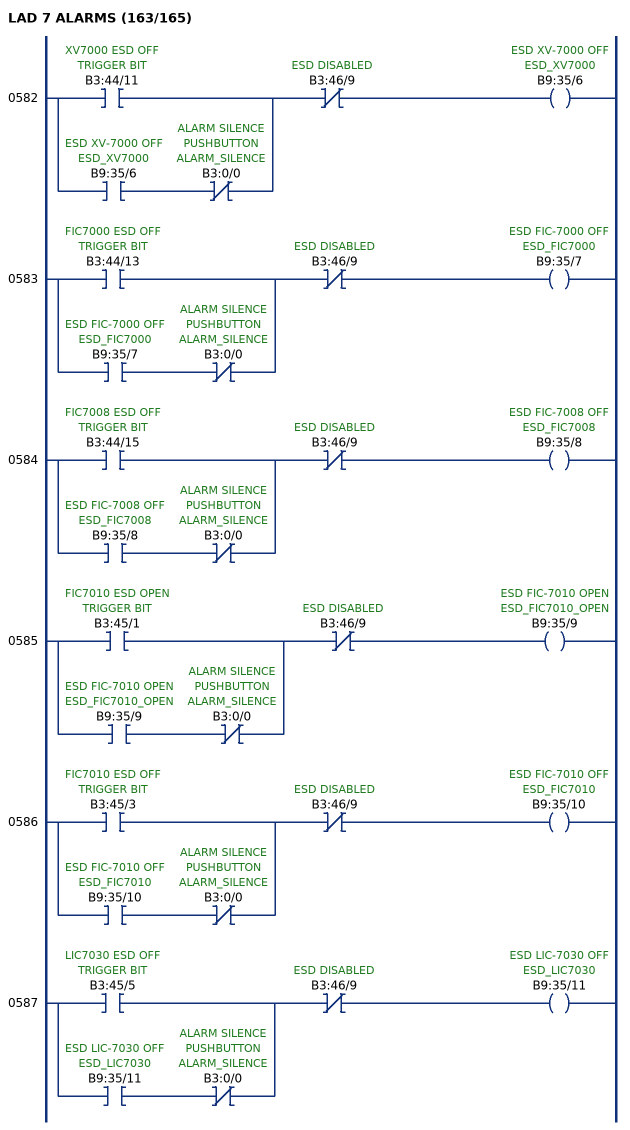
% Rung: 582 %
SOR BST XIC B3:44/11 NXB XIC B9:35/6 XIO B3:0/0 BND XIO B3:46/9 OTE B9:35/6 EOR
%   B3:44/11  "XV7000 ESD OFF TRIGGER BIT" %
%   B9:35/6  ESD_XV7000  "ESD XV-7000 OFF" %
%   B3:0/0  ALARM_SILENCE  "ALARM SILENCE PUSHBUTTON" %
%   B3:46/9  "ESD DISABLED" %
% Rung: 583 %
SOR BST XIC B3:44/13 NXB XIC B9:35/7 XIO B3:0/0 BND XIO B3:46/9 OTE B9:35/7 EOR
%   B3:44/13  "FIC7000 ESD OFF TRIGGER BIT" %
%   B9:35/7  ESD_FIC7000  "ESD FIC-7000 OFF" %
%   B3:0/0  ALARM_SILENCE  "ALARM SILENCE PUSHBUTTON" %
%   B3:46/9  "ESD DISABLED" %
% Rung: 584 %
SOR BST XIC B3:44/15 NXB XIC B9:35/8 XIO B3:0/0 BND XIO B3:46/9 OTE B9:35/8 EOR
%   B3:44/15  "FIC7008 ESD OFF TRIGGER BIT" %
%   B9:35/8  ESD_FIC7008  "ESD FIC-7008 OFF" %
%   B3:0/0  ALARM_SILENCE  "ALARM SILENCE PUSHBUTTON" %
%   B3:46/9  "ESD DISABLED" %
% Rung: 585 %
SOR BST XIC B3:45/1 NXB XIC B9:35/9 XIO B3:0/0 BND XIO B3:46/9 OTE B9:35/9 EOR
%   B3:45/1  "FIC7010 ESD OPEN TRIGGER BIT" %
%   B9:35/9  ESD_FIC7010_OPEN  "ESD FIC-7010 OPEN" %
%   B3:0/0  ALARM_SILENCE  "ALARM SILENCE PUSHBUTTON" %
%   B3:46/9  "ESD DISABLED" %
% Rung: 586 %
SOR BST XIC B3:45/3 NXB XIC B9:35/10 XIO B3:0/0 BND XIO B3:46/9 OTE B9:35/10 EOR
%   B3:45/3  "FIC7010 ESD OFF TRIGGER BIT" %
%   B9:35/10  ESD_FIC7010  "ESD FIC-7010 OFF" %
%   B3:0/0  ALARM_SILENCE  "ALARM SILENCE PUSHBUTTON" %
%   B3:46/9  "ESD DISABLED" %
% Rung: 587 %
SOR BST XIC B3:45/5 NXB XIC B9:35/11 XIO B3:0/0 BND XIO B3:46/9 OTE B9:35/11 EOR
%   B3:45/5  "LIC7030 ESD OFF TRIGGER BIT" %
%   B9:35/11  ESD_LIC7030  "ESD LIC-7030 OFF" %
%   B3:0/0  ALARM_SILENCE  "ALARM SILENCE PUSHBUTTON" %
%   B3:46/9  "ESD DISABLED" %

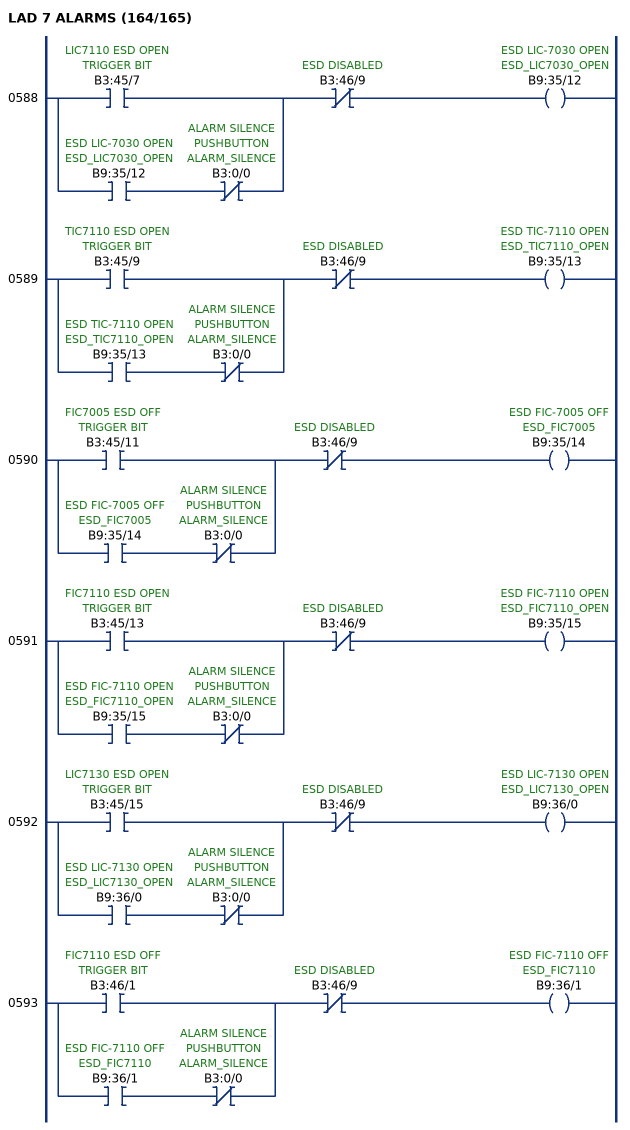
% Rung: 588 %
SOR BST XIC B3:45/7 NXB XIC B9:35/12 XIO B3:0/0 BND XIO B3:46/9 OTE B9:35/12 EOR
%   B3:45/7  "LIC7110 ESD OPEN TRIGGER BIT" %
%   B9:35/12  ESD_LIC7030_OPEN  "ESD LIC-7030 OPEN" %
%   B3:0/0  ALARM_SILENCE  "ALARM SILENCE PUSHBUTTON" %
%   B3:46/9  "ESD DISABLED" %
% Rung: 589 %
SOR BST XIC B3:45/9 NXB XIC B9:35/13 XIO B3:0/0 BND XIO B3:46/9 OTE B9:35/13 EOR
%   B3:45/9  "TIC7110 ESD OPEN TRIGGER BIT" %
%   B9:35/13  ESD_TIC7110_OPEN  "ESD TIC-7110 OPEN" %
%   B3:0/0  ALARM_SILENCE  "ALARM SILENCE PUSHBUTTON" %
%   B3:46/9  "ESD DISABLED" %
% Rung: 590 %
SOR BST XIC B3:45/11 NXB XIC B9:35/14 XIO B3:0/0 BND XIO B3:46/9 OTE B9:35/14 EOR
%   B3:45/11  "FIC7005 ESD OFF TRIGGER BIT" %
%   B9:35/14  ESD_FIC7005  "ESD FIC-7005 OFF" %
%   B3:0/0  ALARM_SILENCE  "ALARM SILENCE PUSHBUTTON" %
%   B3:46/9  "ESD DISABLED" %
% Rung: 591 %
SOR BST XIC B3:45/13 NXB XIC B9:35/15 XIO B3:0/0 BND XIO B3:46/9 OTE B9:35/15 EOR
%   B3:45/13  "FIC7110 ESD OPEN TRIGGER BIT" %
%   B9:35/15  ESD_FIC7110_OPEN  "ESD FIC-7110 OPEN" %
%   B3:0/0  ALARM_SILENCE  "ALARM SILENCE PUSHBUTTON" %
%   B3:46/9  "ESD DISABLED" %
% Rung: 592 %
SOR BST XIC B3:45/15 NXB XIC B9:36/0 XIO B3:0/0 BND XIO B3:46/9 OTE B9:36/0 EOR
%   B3:45/15  "LIC7130 ESD OPEN TRIGGER BIT" %
%   B9:36/0  ESD_LIC7130_OPEN  "ESD LIC-7130 OPEN" %
%   B3:0/0  ALARM_SILENCE  "ALARM SILENCE PUSHBUTTON" %
%   B3:46/9  "ESD DISABLED" %
% Rung: 593 %
SOR BST XIC B3:46/1 NXB XIC B9:36/1 XIO B3:0/0 BND XIO B3:46/9 OTE B9:36/1 EOR
%   B3:46/1  "FIC7110 ESD OFF TRIGGER BIT" %
%   B9:36/1  ESD_FIC7110  "ESD FIC-7110 OFF" %
%   B3:0/0  ALARM_SILENCE  "ALARM SILENCE PUSHBUTTON" %
%   B3:46/9  "ESD DISABLED" %

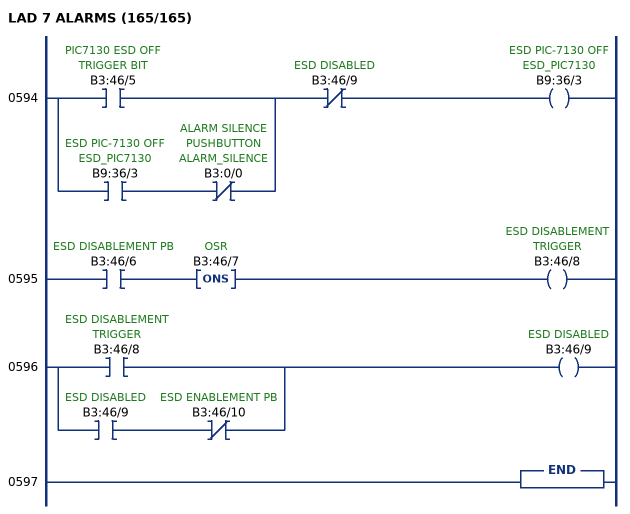
% Rung: 594 %
SOR BST XIC B3:46/5 NXB XIC B9:36/3 XIO B3:0/0 BND XIO B3:46/9 OTE B9:36/3 EOR
%   B3:46/5  "PIC7130 ESD OFF TRIGGER BIT" %
%   B9:36/3  ESD_PIC7130  "ESD PIC-7130 OFF" %
%   B3:0/0  ALARM_SILENCE  "ALARM SILENCE PUSHBUTTON" %
%   B3:46/9  "ESD DISABLED" %
% Rung: 595 %
SOR XIC B3:46/6 OSR B3:46/7 OTE B3:46/8 EOR
%   B3:46/6  "ESD DISABLEMENT PB" %
%   B3:46/7  "OSR" %
%   B3:46/8  "ESD DISABLEMENT TRIGGER" %
% Rung: 596 %
SOR BST XIC B3:46/8 NXB XIC B3:46/9 XIO B3:46/10 BND OTE B3:46/9 EOR
%   B3:46/8  "ESD DISABLEMENT TRIGGER" %
%   B3:46/9  "ESD DISABLED" %
%   B3:46/10  "ESD ENABLEMENT PB" %
% Rung: 597 %
SOR END EOR

LADDER 8 "HMI IO"
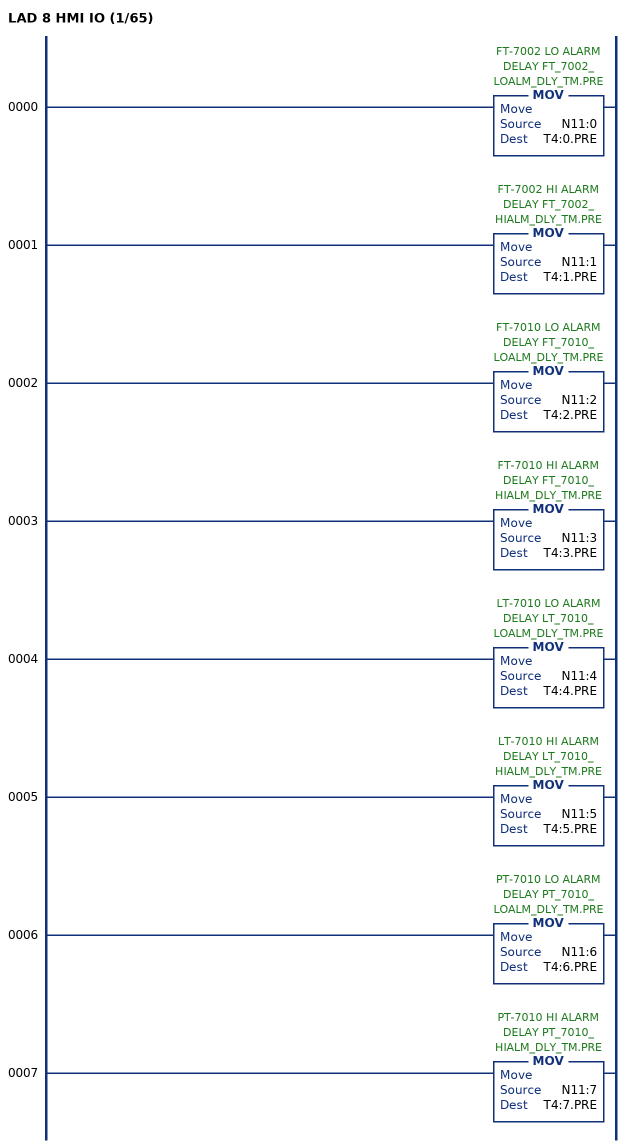
% Rung: 0 %
SOR MOV N11:0 T4:0.PRE EOR
%   N11:0  FT_7002_LOALM_DLY_SP  "FT-7002 LO ALARM DELAY SP FROM HMI" %
%   T4:0  FT_7002_LOALM_DLY_TM  "FT-7002 LO ALARM DELAY" %
% Rung: 1 %
SOR MOV N11:1 T4:1.PRE EOR
%   N11:1  FT_7002_HIALM_DLY_SP  "FT-7002 HI ALARM DELAY SP FROM HMI" %
%   T4:1  FT_7002_HIALM_DLY_TM  "FT-7002 HI ALARM DELAY" %
% Rung: 2 %
SOR MOV N11:2 T4:2.PRE EOR
%   N11:2  FT_7010_LOALM_DLY_SP  "FT-7010 LO ALARM DELAY SP FROM HMI" %
%   T4:2  FT_7010_LOALM_DLY_TM  "FT-7010 LO ALARM DELAY" %
% Rung: 3 %
SOR MOV N11:3 T4:3.PRE EOR
%   N11:3  FT_7010_HIALM_DLY_SP  "FT-7010 HI ALARM DELAY SP FROM HMI" %
%   T4:3  FT_7010_HIALM_DLY_TM  "FT-7010 HI ALARM DELAY" %
% Rung: 4 %
SOR MOV N11:4 T4:4.PRE EOR
%   N11:4  LT_7010_LOALM_DLY_SP  "LT-7010 LO ALARM DELAY SP FROM HMI" %
%   T4:4  LT_7010_LOALM_DLY_TM  "LT-7010 LO ALARM DELAY" %
% Rung: 5 %
SOR MOV N11:5 T4:5.PRE EOR
%   N11:5  LT_7010_HIALM_DLY_SP  "LT-7010 HI ALARM DELAY SP FROM HMI" %
%   T4:5  LT_7010_HIALM_DLY_TM  "LT-7010 HI ALARM DELAY" %
% Rung: 6 %
SOR MOV N11:6 T4:6.PRE EOR
%   N11:6  PT_7010_LOALM_DLY_SP  "PT-7010 LO ALARM DELAY SP FROM HMI" %
%   T4:6  PT_7010_LOALM_DLY_TM  "PT-7010 LO ALARM DELAY" %
% Rung: 7 %
SOR MOV N11:7 T4:7.PRE EOR
%   N11:7  PT_7010_HIALM_DLY_SP  "PT-7010 HI ALARM DELAY SP FROM HMI" %
%   T4:7  PT_7010_HIALM_DLY_TM  "PT-7010 HI ALARM DELAY" %

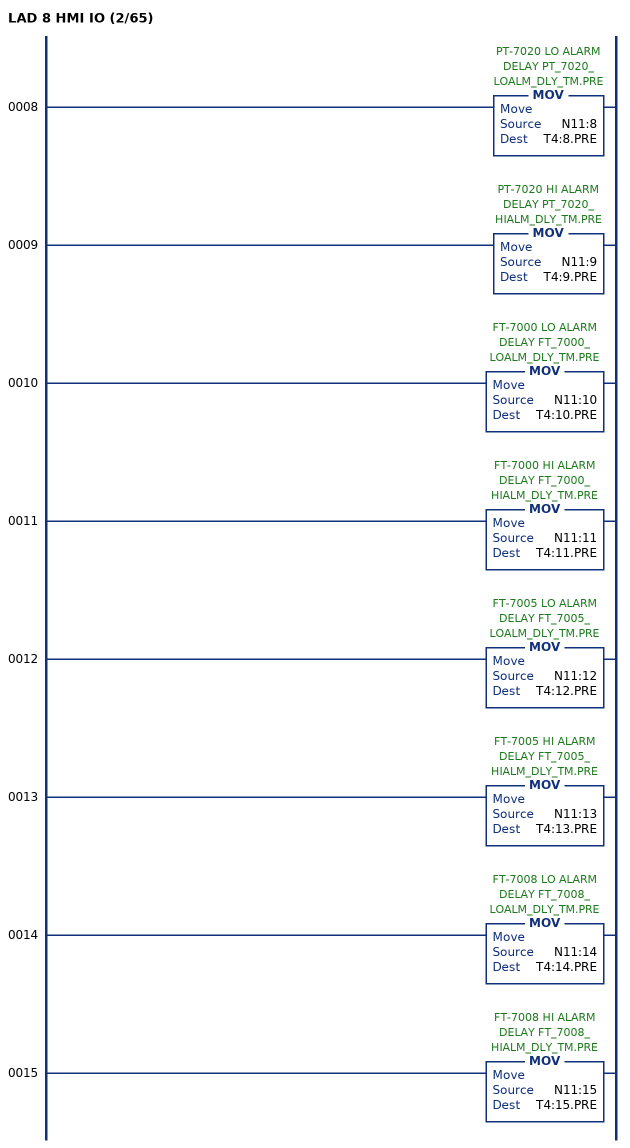
% Rung: 8 %
SOR MOV N11:8 T4:8.PRE EOR
%   N11:8  PT_7020_LOALM_DLY_SP  "PT-7020 LO ALARM DELAY SP FROM HMI" %
%   T4:8  PT_7020_LOALM_DLY_TM  "PT-7020 LO ALARM DELAY" %
% Rung: 9 %
SOR MOV N11:9 T4:9.PRE EOR
%   N11:9  PT_7020_HIALM_DLY_SP  "PT-7020 HI ALARM DELAY SP FROM HMI" %
%   T4:9  PT_7020_HIALM_DLY_TM  "PT-7020 HI ALARM DELAY" %
% Rung: 10 %
SOR MOV N11:10 T4:10.PRE EOR
%   N11:10  FT_7000_LOALM_DLY_SP  "FT-7000 LO ALARM DELAY SP FROM HMI" %
%   T4:10  FT_7000_LOALM_DLY_TM  "FT-7000 LO ALARM DELAY" %
% Rung: 11 %
SOR MOV N11:11 T4:11.PRE EOR
%   N11:11  FT_7000_HIALM_DLY_SP  "FT-7000 HI ALARM DELAY SP FROM HMI" %
%   T4:11  FT_7000_HIALM_DLY_TM  "FT-7000 HI ALARM DELAY" %
% Rung: 12 %
SOR MOV N11:12 T4:12.PRE EOR
%   N11:12  FT_7005_LOALM_DLY_SP  "FT-7005 LO ALARM DELAY SP FROM HMI" %
%   T4:12  FT_7005_LOALM_DLY_TM  "FT-7005 LO ALARM DELAY" %
% Rung: 13 %
SOR MOV N11:13 T4:13.PRE EOR
%   N11:13  FT_7005_HIALM_DLY_SP  "FT-7005 HI ALARM DELAY SP FROM HMI" %
%   T4:13  FT_7005_HIALM_DLY_TM  "FT-7005 HI ALARM DELAY" %
% Rung: 14 %
SOR MOV N11:14 T4:14.PRE EOR
%   N11:14  FT_7008_LOALM_DLY_SP  "FT-7008 LO ALARM DELAY SP FROM HMI" %
%   T4:14  FT_7008_LOALM_DLY_TM  "FT-7008 LO ALARM DELAY" %
% Rung: 15 %
SOR MOV N11:15 T4:15.PRE EOR
%   N11:15  FT_7008_HIALM_DLY_SP  "FT-7008 HI ALARM DELAY SP FROM HMI" %
%   T4:15  FT_7008_HIALM_DLY_TM  "FT-7008 HI ALARM DELAY" %

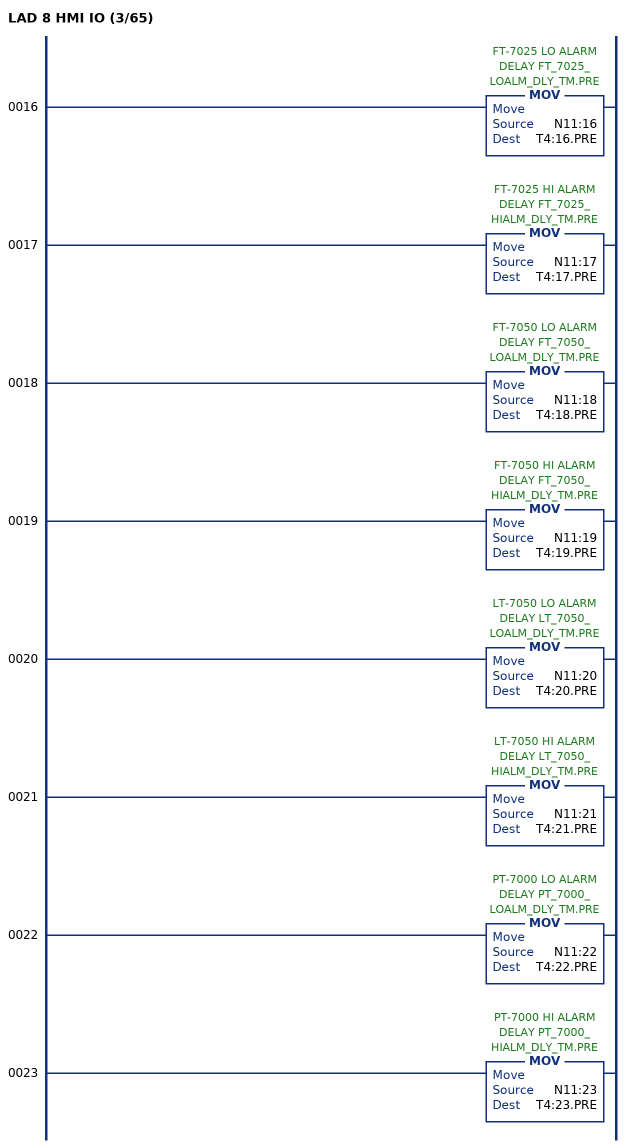
% Rung: 16 %
SOR MOV N11:16 T4:16.PRE EOR
%   N11:16  FT_7025_LOALM_DLY_SP  "FT-7025 LO ALARM DELAY SP FROM HMI" %
%   T4:16  FT_7025_LOALM_DLY_TM  "FT-7025 LO ALARM DELAY" %
% Rung: 17 %
SOR MOV N11:17 T4:17.PRE EOR
%   N11:17  FT_7025_HIALM_DLY_SP  "FT-7025 HI ALARM DELAY SP FROM HMI" %
%   T4:17  FT_7025_HIALM_DLY_TM  "FT-7025 HI ALARM DELAY" %
% Rung: 18 %
SOR MOV N11:18 T4:18.PRE EOR
%   N11:18  FT_7050_LOALM_DLY_SP  "FT-7050 LO ALARM DELAY SP FROM HMI" %
%   T4:18  FT_7050_LOALM_DLY_TM  "FT-7050 LO ALARM DELAY" %
% Rung: 19 %
SOR MOV N11:19 T4:19.PRE EOR
%   N11:19  FT_7050_HIALM_DLY_SP  "FT-7050 HI ALARM DELAY SP FROM HMI" %
%   T4:19  FT_7050_HIALM_DLY_TM  "FT-7050 HI ALARM DELAY" %
% Rung: 20 %
SOR MOV N11:20 T4:20.PRE EOR
%   N11:20  LT_7050_LOALM_DLY_SP  "LT-7050 LO ALARM DELAY SP FROM HMI" %
%   T4:20  LT_7050_LOALM_DLY_TM  "LT-7050 LO ALARM DELAY" %
% Rung: 21 %
SOR MOV N11:21 T4:21.PRE EOR
%   N11:21  LT_7050_HIALM_DLY_SP  "LT-7050 HI ALARM DELAY SP FROM HMI" %
%   T4:21  LT_7050_HIALM_DLY_TM  "LT-7050 HI ALARM DELAY" %
% Rung: 22 %
SOR MOV N11:22 T4:22.PRE EOR
%   N11:22  PT_7000_LOALM_DLY_SP  "PT-7000 LO ALARM DELAY SP FROM HMI" %
%   T4:22  PT_7000_LOALM_DLY_TM  "PT-7000 LO ALARM DELAY" %
% Rung: 23 %
SOR MOV N11:23 T4:23.PRE EOR
%   N11:23  PT_7000_HIALM_DLY_SP  "PT-7000 HI ALARM DELAY SP FROM HMI" %
%   T4:23  PT_7000_HIALM_DLY_TM  "PT-7000 HI ALARM DELAY" %

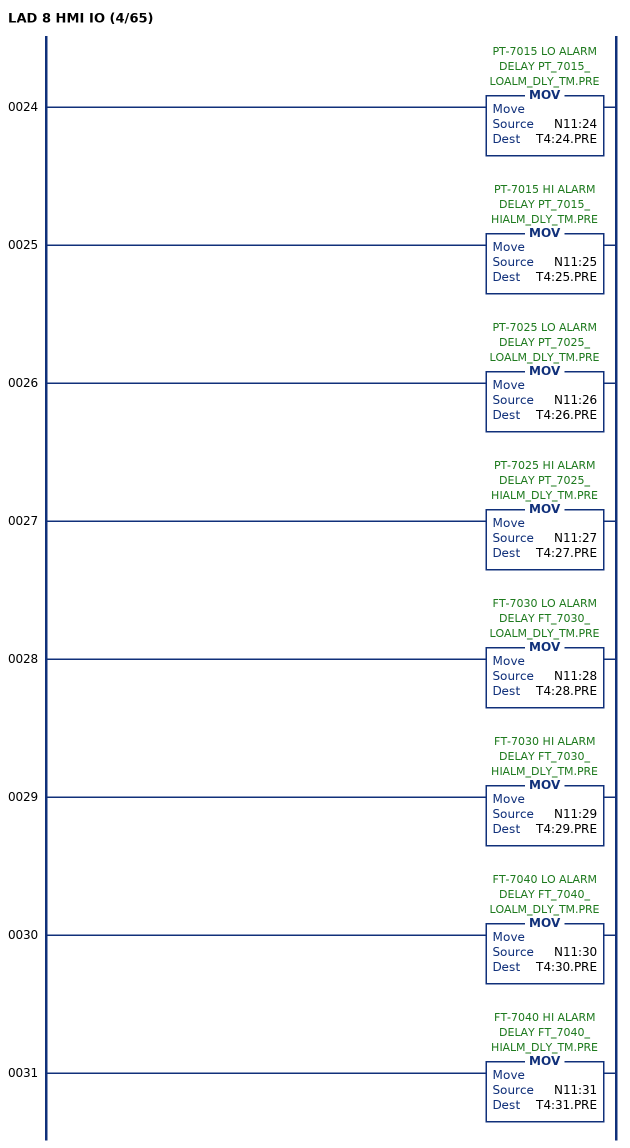
% Rung: 24 %
SOR MOV N11:24 T4:24.PRE EOR
%   N11:24  PT_7015_LOALM_DLY_SP  "PT-7015 LO ALARM DELAY SP FROM HMI" %
%   T4:24  PT_7015_LOALM_DLY_TM  "PT-7015 LO ALARM DELAY" %
% Rung: 25 %
SOR MOV N11:25 T4:25.PRE EOR
%   N11:25  PT_7015_HIALM_DLY_SP  "PT-7015 HI ALARM DELAY SP FROM HMI" %
%   T4:25  PT_7015_HIALM_DLY_TM  "PT-7015 HI ALARM DELAY" %
% Rung: 26 %
SOR MOV N11:26 T4:26.PRE EOR
%   N11:26  PT_7025_LOALM_DLY_SP  "PT-7025 LO ALARM DELAY SP FROM HMI" %
%   T4:26  PT_7025_LOALM_DLY_TM  "PT-7025 LO ALARM DELAY" %
% Rung: 27 %
SOR MOV N11:27 T4:27.PRE EOR
%   N11:27  PT_7025_HIALM_DLY_SP  "PT-7025 HI ALARM DELAY SP FROM HMI" %
%   T4:27  PT_7025_HIALM_DLY_TM  "PT-7025 HI ALARM DELAY" %
% Rung: 28 %
SOR MOV N11:28 T4:28.PRE EOR
%   N11:28  FT_7030_LOALM_DLY_SP  "FT-7030 LO ALARM DELAY SP FROM HMI" %
%   T4:28  FT_7030_LOALM_DLY_TM  "FT-7030 LO ALARM DELAY" %
% Rung: 29 %
SOR MOV N11:29 T4:29.PRE EOR
%   N11:29  FT_7030_HIALM_DLY_SP  "FT-7030 HI ALARM DELAY SP FROM HMI" %
%   T4:29  FT_7030_HIALM_DLY_TM  "FT-7030 HI ALARM DELAY" %
% Rung: 30 %
SOR MOV N11:30 T4:30.PRE EOR
%   N11:30  FT_7040_LOALM_DLY_SP  "FT-7040 LO ALARM DELAY SP FROM HMI" %
%   T4:30  FT_7040_LOALM_DLY_TM  "FT-7040 LO ALARM DELAY" %
% Rung: 31 %
SOR MOV N11:31 T4:31.PRE EOR
%   N11:31  FT_7040_HIALM_DLY_SP  "FT-7040 HI ALARM DELAY SP FROM HMI" %
%   T4:31  FT_7040_HIALM_DLY_TM  "FT-7040 HI ALARM DELAY" %

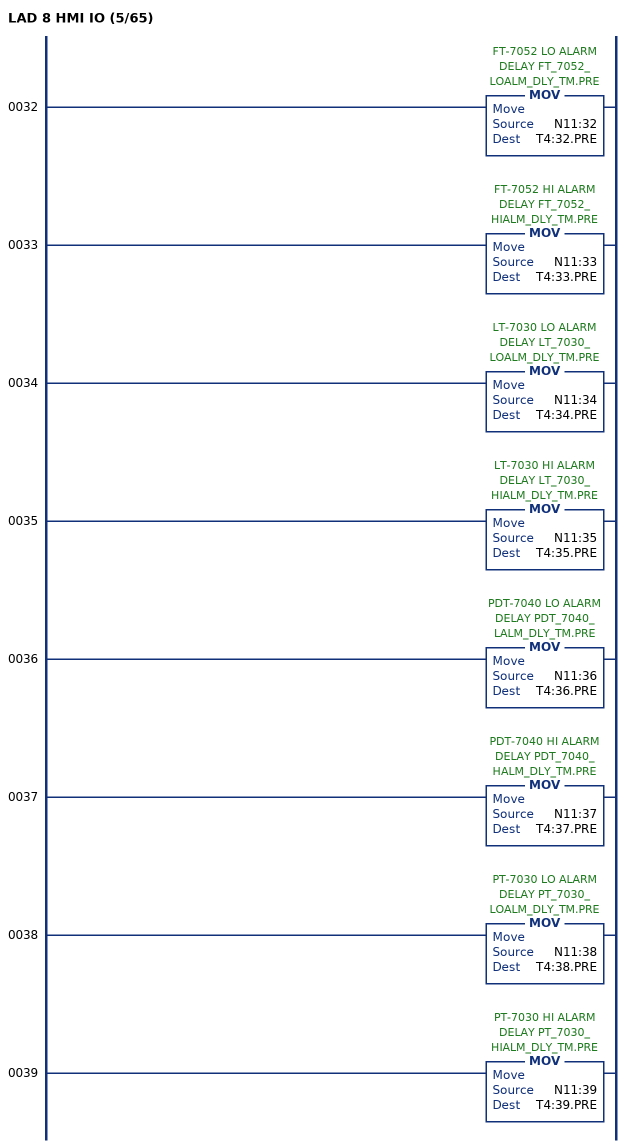
% Rung: 32 %
SOR MOV N11:32 T4:32.PRE EOR
%   N11:32  FT_7052_LOALM_DLY_SP  "FT-7052 LO ALARM DELAY SP FROM HMI" %
%   T4:32  FT_7052_LOALM_DLY_TM  "FT-7052 LO ALARM DELAY" %
% Rung: 33 %
SOR MOV N11:33 T4:33.PRE EOR
%   N11:33  FT_7052_HIALM_DLY_SP  "FT-7052 HI ALARM DELAY SP FROM HMI" %
%   T4:33  FT_7052_HIALM_DLY_TM  "FT-7052 HI ALARM DELAY" %
% Rung: 34 %
SOR MOV N11:34 T4:34.PRE EOR
%   N11:34  LT_7030_LOALM_DLY_SP  "LT-7030 LO ALARM DELAY SP FROM HMI" %
%   T4:34  LT_7030_LOALM_DLY_TM  "LT-7030 LO ALARM DELAY" %
% Rung: 35 %
SOR MOV N11:35 T4:35.PRE EOR
%   N11:35  LT_7030_HIALM_DLY_SP  "LT-7030 HI ALARM DELAY SP FROM HMI" %
%   T4:35  LT_7030_HIALM_DLY_TM  "LT-7030 HI ALARM DELAY" %
% Rung: 36 %
SOR MOV N11:36 T4:36.PRE EOR
%   N11:36  PDT_7040_LALM_DLY_SP  "PDT-7040 LO ALARM DELAY SP FROM HMI" %
%   T4:36  PDT_7040_LALM_DLY_TM  "PDT-7040 LO ALARM DELAY" %
% Rung: 37 %
SOR MOV N11:37 T4:37.PRE EOR
%   N11:37  PDT_7040_HALM_DLY_SP  "PDT-7040 HI ALARM DELAY SP FROM HMI" %
%   T4:37  PDT_7040_HALM_DLY_TM  "PDT-7040 HI ALARM DELAY" %
% Rung: 38 %
SOR MOV N11:38 T4:38.PRE EOR
%   N11:38  PT_7030_LOALM_DLY_SP  "PT-7030 LO ALARM DELAY SP FROM HMI" %
%   T4:38  PT_7030_LOALM_DLY_TM  "PT-7030 LO ALARM DELAY" %
% Rung: 39 %
SOR MOV N11:39 T4:39.PRE EOR
%   N11:39  PT_7030_HIALM_DLY_SP  "PT-7030 HI ALARM DELAY SP FROM HMI" %
%   T4:39  PT_7030_HIALM_DLY_TM  "PT-7030 HI ALARM DELAY" %

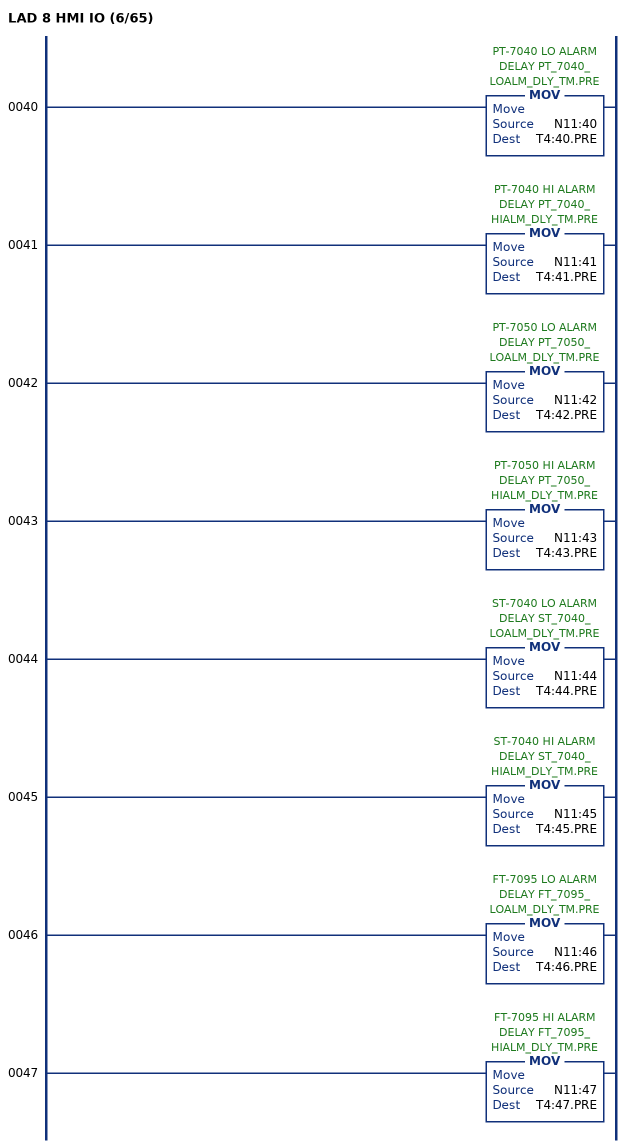
% Rung: 40 %
SOR MOV N11:40 T4:40.PRE EOR
%   N11:40  PT_7040_LOALM_DLY_SP  "PT-7040 LO ALARM DELAY SP FROM HMI" %
%   T4:40  PT_7040_LOALM_DLY_TM  "PT-7040 LO ALARM DELAY" %
% Rung: 41 %
SOR MOV N11:41 T4:41.PRE EOR
%   N11:41  PT_7040_HIALM_DLY_SP  "PT-7040 HI ALARM DELAY SP FROM HMI" %
%   T4:41  PT_7040_HIALM_DLY_TM  "PT-7040 HI ALARM DELAY" %
% Rung: 42 %
SOR MOV N11:42 T4:42.PRE EOR
%   N11:42  PT_7050_LOALM_DLY_SP  "PT-7050 LO ALARM DELAY SP FROM HMI" %
%   T4:42  PT_7050_LOALM_DLY_TM  "PT-7050 LO ALARM DELAY" %
% Rung: 43 %
SOR MOV N11:43 T4:43.PRE EOR
%   N11:43  PT_7050_HIALM_DLY_SP  "PT-7050 HI ALARM DELAY SP FROM HMI" %
%   T4:43  PT_7050_HIALM_DLY_TM  "PT-7050 HI ALARM DELAY" %
% Rung: 44 %
SOR MOV N11:44 T4:44.PRE EOR
%   N11:44  ST_7040_LOALM_DLY_SP  "ST-7040 LO ALARM DELAY SP FROM HMI" %
%   T4:44  ST_7040_LOALM_DLY_TM  "ST-7040 LO ALARM DELAY" %
% Rung: 45 %
SOR MOV N11:45 T4:45.PRE EOR
%   N11:45  ST_7040_HIALM_DLY_SP  "ST-7040 HI ALARM DELAY SP FROM HMI" %
%   T4:45  ST_7040_HIALM_DLY_TM  "ST-7040 HI ALARM DELAY" %
% Rung: 46 %
SOR MOV N11:46 T4:46.PRE EOR
%   N11:46  FT_7095_LOALM_DLY_SP  "FT-7095 LO ALARM DELAY SP FROM HMI" %
%   T4:46  FT_7095_LOALM_DLY_TM  "FT-7095 LO ALARM DELAY" %
% Rung: 47 %
SOR MOV N11:47 T4:47.PRE EOR
%   N11:47  FT_7095_HIALM_DLY_SP  "FT-7095 HI ALARM DELAY SP FROM HMI" %
%   T4:47  FT_7095_HIALM_DLY_TM  "FT-7095 HI ALARM DELAY" %

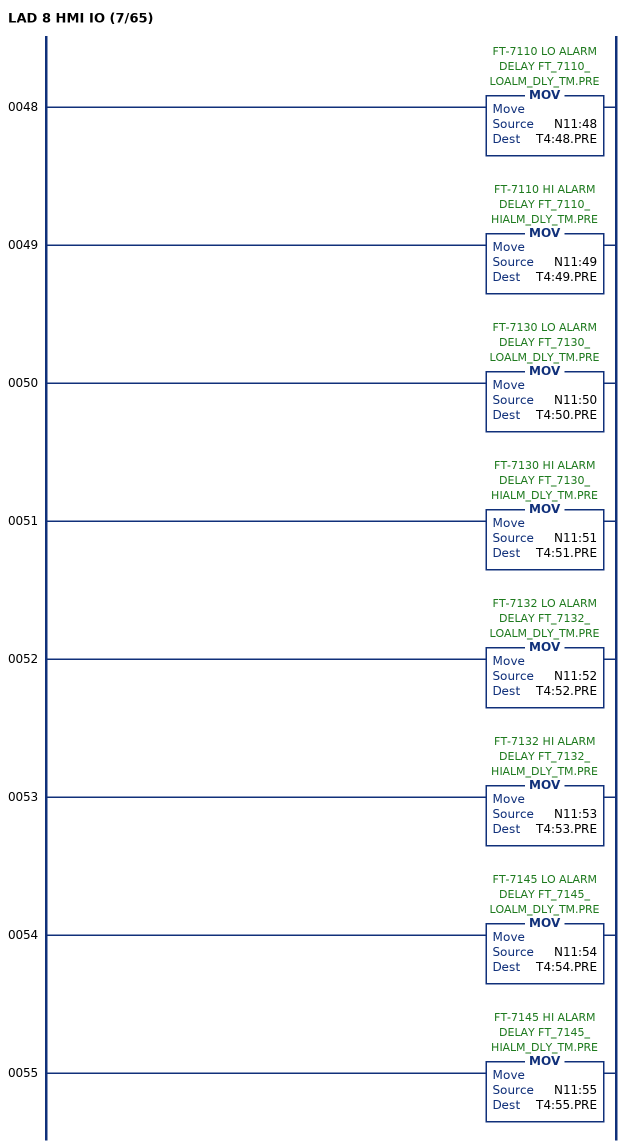
% Rung: 48 %
SOR MOV N11:48 T4:48.PRE EOR
%   N11:48  FT_7110_LOALM_DLY_SP  "FT-7110 LO ALARM DELAY SP FROM HMI" %
%   T4:48  FT_7110_LOALM_DLY_TM  "FT-7110 LO ALARM DELAY" %
% Rung: 49 %
SOR MOV N11:49 T4:49.PRE EOR
%   N11:49  FT_7110_HIALM_DLY_SP  "FT-7110 HI ALARM DELAY SP FROM HMI" %
%   T4:49  FT_7110_HIALM_DLY_TM  "FT-7110 HI ALARM DELAY" %
% Rung: 50 %
SOR MOV N11:50 T4:50.PRE EOR
%   N11:50  FT_7130_LOALM_DLY_SP  "FT-7130 LO ALARM DELAY SP FROM HMI" %
%   T4:50  FT_7130_LOALM_DLY_TM  "FT-7130 LO ALARM DELAY" %
% Rung: 51 %
SOR MOV N11:51 T4:51.PRE EOR
%   N11:51  FT_7130_HIALM_DLY_SP  "FT-7130 HI ALARM DELAY SP FROM HMI" %
%   T4:51  FT_7130_HIALM_DLY_TM  "FT-7130 HI ALARM DELAY" %
% Rung: 52 %
SOR MOV N11:52 T4:52.PRE EOR
%   N11:52  FT_7132_LOALM_DLY_SP  "FT-7132 LO ALARM DELAY SP FROM HMI" %
%   T4:52  FT_7132_LOALM_DLY_TM  "FT-7132 LO ALARM DELAY" %
% Rung: 53 %
SOR MOV N11:53 T4:53.PRE EOR
%   N11:53  FT_7132_HIALM_DLY_SP  "FT-7132 HI ALARM DELAY SP FROM HMI" %
%   T4:53  FT_7132_HIALM_DLY_TM  "FT-7132 HI ALARM DELAY" %
% Rung: 54 %
SOR MOV N11:54 T4:54.PRE EOR
%   N11:54  FT_7145_LOALM_DLY_SP  "FT-7145 LO ALARM DELAY SP FROM HMI" %
%   T4:54  FT_7145_LOALM_DLY_TM  "FT-7145 LO ALARM DELAY" %
% Rung: 55 %
SOR MOV N11:55 T4:55.PRE EOR
%   N11:55  FT_7145_HIALM_DLY_SP  "FT-7145 HI ALARM DELAY SP FROM HMI" %
%   T4:55  FT_7145_HIALM_DLY_TM  "FT-7145 HI ALARM DELAY" %

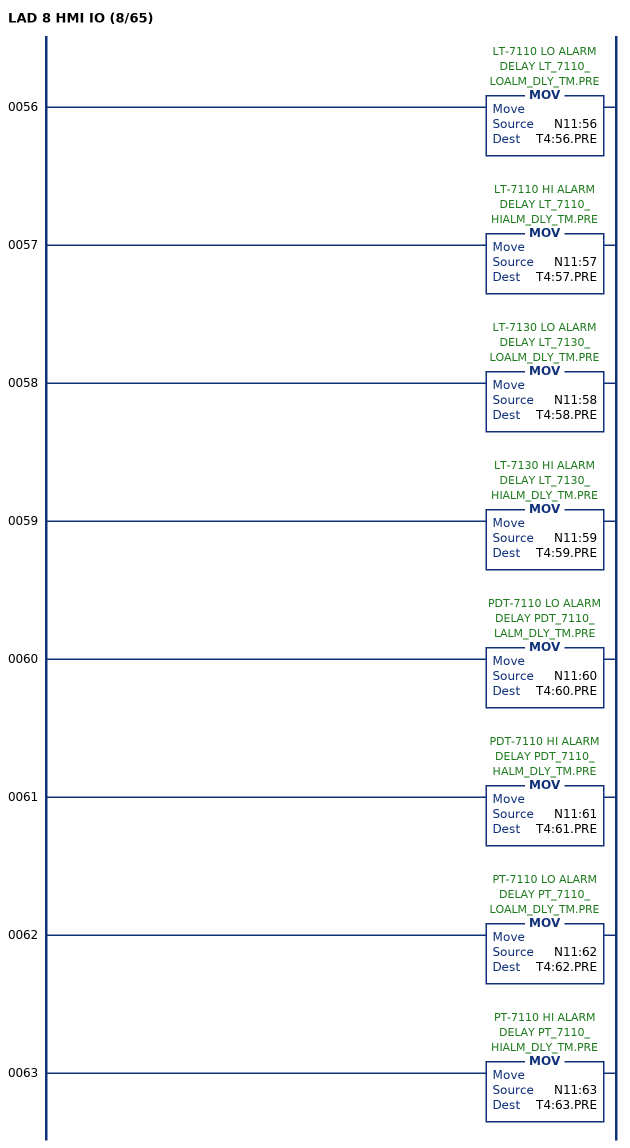
% Rung: 56 %
SOR MOV N11:56 T4:56.PRE EOR
%   N11:56  LT_7110_LOALM_DLY_SP  "LT-7110 LO ALARM DELAY SP FROM HMI" %
%   T4:56  LT_7110_LOALM_DLY_TM  "LT-7110 LO ALARM DELAY" %
% Rung: 57 %
SOR MOV N11:57 T4:57.PRE EOR
%   N11:57  LT_7110_HIALM_DLY_SP  "LT-7110 HI ALARM DELAY SP FROM HMI" %
%   T4:57  LT_7110_HIALM_DLY_TM  "LT-7110 HI ALARM DELAY" %
% Rung: 58 %
SOR MOV N11:58 T4:58.PRE EOR
%   N11:58  LT_7130_LOALM_DLY_SP  "LT-7130 LO ALARM DELAY SP FROM HMI" %
%   T4:58  LT_7130_LOALM_DLY_TM  "LT-7130 LO ALARM DELAY" %
% Rung: 59 %
SOR MOV N11:59 T4:59.PRE EOR
%   N11:59  LT_7130_HIALM_DLY_SP  "LT-7130 HI ALARM DELAY SP FROM HMI" %
%   T4:59  LT_7130_HIALM_DLY_TM  "LT-7130 HI ALARM DELAY" %
% Rung: 60 %
SOR MOV N11:60 T4:60.PRE EOR
%   N11:60  PDT_7110_LALM_DLY_SP  "PDT-7110 LO ALARM DELAY SP FROM HMI" %
%   T4:60  PDT_7110_LALM_DLY_TM  "PDT-7110 LO ALARM DELAY" %
% Rung: 61 %
SOR MOV N11:61 T4:61.PRE EOR
%   N11:61  PDT_7110_HALM_DLY_SP  "PDT-7110 HI ALARM DELAY SP FROM HMI" %
%   T4:61  PDT_7110_HALM_DLY_TM  "PDT-7110 HI ALARM DELAY" %
% Rung: 62 %
SOR MOV N11:62 T4:62.PRE EOR
%   N11:62  PT_7110_LOALM_DLY_SP  "PT-7110 LO ALARM DELAY SP FROM HMI" %
%   T4:62  PT_7110_LOALM_DLY_TM  "PT-7110 LO ALARM DELAY" %
% Rung: 63 %
SOR MOV N11:63 T4:63.PRE EOR
%   N11:63  PT_7110_HIALM_DLY_SP  "PT-7110 HI ALARM DELAY SP FROM HMI" %
%   T4:63  PT_7110_HIALM_DLY_TM  "PT-7110 HI ALARM DELAY" %

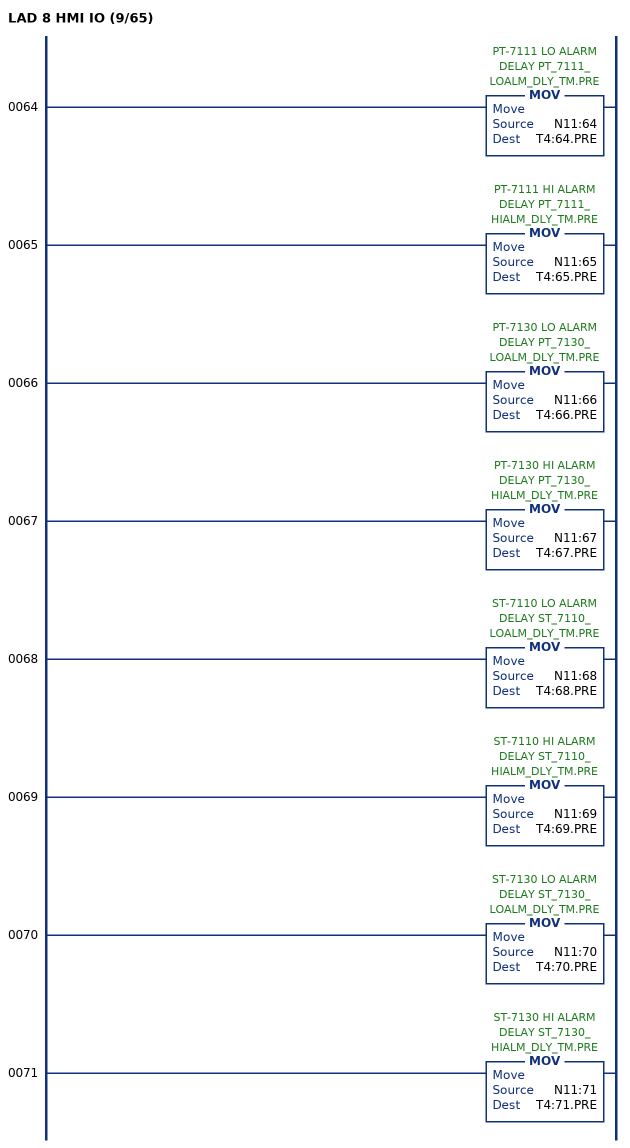
% Rung: 64 %
SOR MOV N11:64 T4:64.PRE EOR
%   N11:64  PT_7111_LOALM_DLY_SP  "PT-7111 LO ALARM DELAY SP FROM HMI" %
%   T4:64  PT_7111_LOALM_DLY_TM  "PT-7111 LO ALARM DELAY" %
% Rung: 65 %
SOR MOV N11:65 T4:65.PRE EOR
%   N11:65  PT_7111_HIALM_DLY_SP  "PT-7111 HI ALARM DELAY SP FROM HMI" %
%   T4:65  PT_7111_HIALM_DLY_TM  "PT-7111 HI ALARM DELAY" %
% Rung: 66 %
SOR MOV N11:66 T4:66.PRE EOR
%   N11:66  PT_7130_LOALM_DLY_SP  "PT-7130 LO ALARM DELAY SP FROM HMI" %
%   T4:66  PT_7130_LOALM_DLY_TM  "PT-7130 LO ALARM DELAY" %
% Rung: 67 %
SOR MOV N11:67 T4:67.PRE EOR
%   N11:67  PT_7130_HIALM_DLY_SP  "PT-7130 HI ALARM DELAY SP FROM HMI" %
%   T4:67  PT_7130_HIALM_DLY_TM  "PT-7130 HI ALARM DELAY" %
% Rung: 68 %
SOR MOV N11:68 T4:68.PRE EOR
%   N11:68  ST_7110_LOALM_DLY_SP  "ST-7110 LO ALARM DELAY SP FROM HMI" %
%   T4:68  ST_7110_LOALM_DLY_TM  "ST-7110 LO ALARM DELAY" %
% Rung: 69 %
SOR MOV N11:69 T4:69.PRE EOR
%   N11:69  ST_7110_HIALM_DLY_SP  "ST-7110 HI ALARM DELAY SP FROM HMI" %
%   T4:69  ST_7110_HIALM_DLY_TM  "ST-7110 HI ALARM DELAY" %
% Rung: 70 %
SOR MOV N11:70 T4:70.PRE EOR
%   N11:70  ST_7130_LOALM_DLY_SP  "ST-7130 LO ALARM DELAY SP FROM HMI" %
%   T4:70  ST_7130_LOALM_DLY_TM  "ST-7130 LO ALARM DELAY" %
% Rung: 71 %
SOR MOV N11:71 T4:71.PRE EOR
%   N11:71  ST_7130_HIALM_DLY_SP  "ST-7130 HI ALARM DELAY SP FROM HMI" %
%   T4:71  ST_7130_HIALM_DLY_TM  "ST-7130 HI ALARM DELAY" %

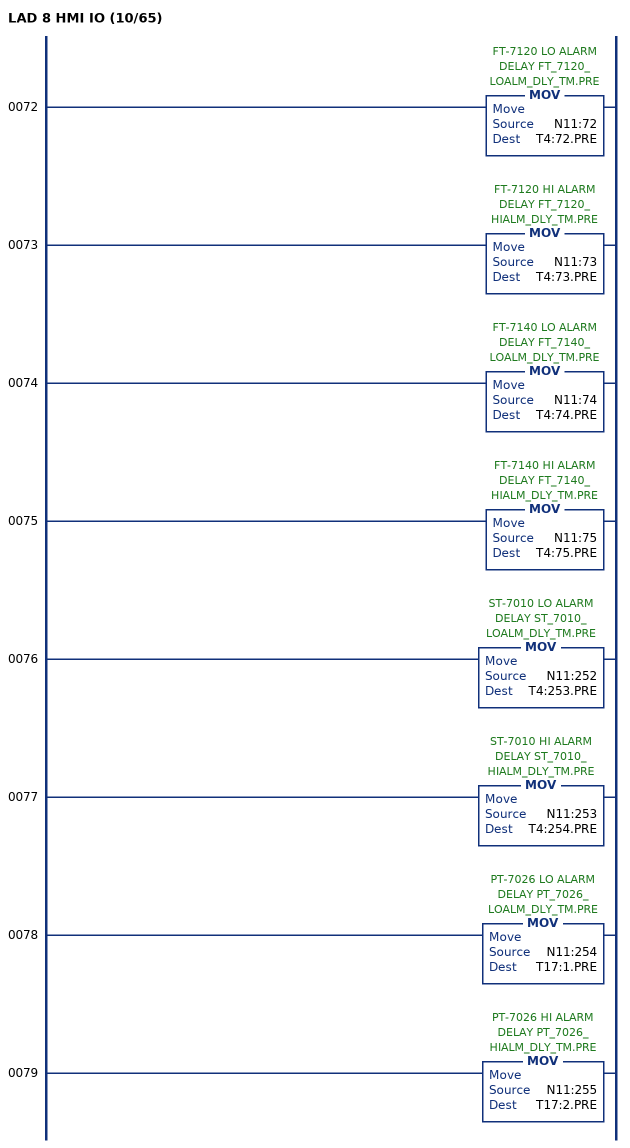
% Rung: 72 %
SOR MOV N11:72 T4:72.PRE EOR
%   N11:72  FT_7120_LOALM_DLY_SP  "FT-7120 LO ALARM DELAY SP FROM HMI" %
%   T4:72  FT_7120_LOALM_DLY_TM  "FT-7120 LO ALARM DELAY" %
% Rung: 73 %
SOR MOV N11:73 T4:73.PRE EOR
%   N11:73  FT_7120_HIALM_DLY_SP  "FT-7120 HI ALARM DELAY SP FROM HMI" %
%   T4:73  FT_7120_HIALM_DLY_TM  "FT-7120 HI ALARM DELAY" %
% Rung: 74 %
SOR MOV N11:74 T4:74.PRE EOR
%   N11:74  FT_7140_LOALM_DLY_SP  "FT-7140 LO ALARM DELAY SP FROM HMI" %
%   T4:74  FT_7140_LOALM_DLY_TM  "FT-7140 LO ALARM DELAY" %
% Rung: 75 %
SOR MOV N11:75 T4:75.PRE EOR
%   N11:75  FT_7140_HIALM_DLY_SP  "FT-7140 HI ALARM DELAY SP FROM HMI" %
%   T4:75  FT_7140_HIALM_DLY_TM  "FT-7140 HI ALARM DELAY" %
% Rung: 76 %
SOR MOV N11:252 T4:253.PRE EOR
%   N11:252  ST_7010_LOALM_DLY_SP  "ST-7010 LO ALARM DELAY SP FROM HMI" %
%   T4:253  ST_7010_LOALM_DLY_TM  "ST-7010 LO ALARM DELAY" %
% Rung: 77 %
SOR MOV N11:253 T4:254.PRE EOR
%   N11:253  ST_7010_HIALM_DLY_SP  "ST-7010 HI ALARM DELAY SP FROM HMI" %
%   T4:254  ST_7010_HIALM_DLY_TM  "ST-7010 HI ALARM DELAY" %
% Rung: 78 %
SOR MOV N11:254 T17:1.PRE EOR
%   N11:254  PT_7026_LOALM_DLY_SP  "PT-7026 LO ALARM DELAY SP FROM HMI" %
%   T17:1  PT_7026_LOALM_DLY_TM  "PT-7026 LO ALARM DELAY" %
% Rung: 79 %
SOR MOV N11:255 T17:2.PRE EOR
%   N11:255  PT_7026_HIALM_DLY_SP  "PT-7026 HI ALARM DELAY SP FROM HMI" %
%   T17:2  PT_7026_HIALM_DLY_TM  "PT-7026 HI ALARM DELAY" %

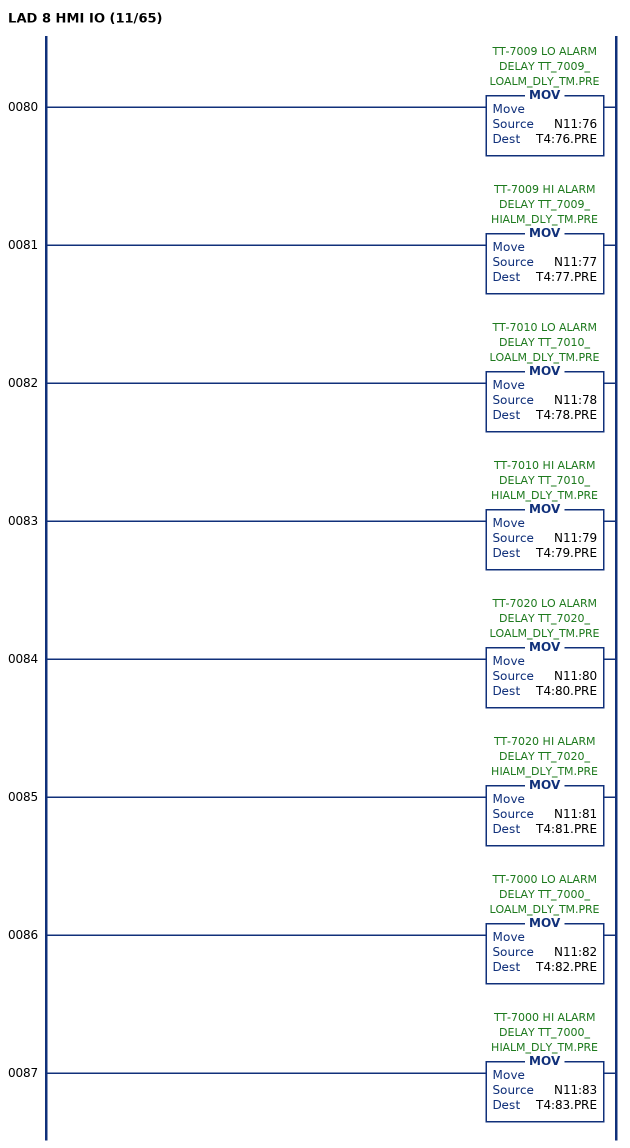
% Rung: 80 %
SOR MOV N11:76 T4:76.PRE EOR
%   N11:76  TT_7009_LOALM_DLY_SP  "TT-7009 LO ALARM DELAY SP FROM HMI" %
%   T4:76  TT_7009_LOALM_DLY_TM  "TT-7009 LO ALARM DELAY" %
% Rung: 81 %
SOR MOV N11:77 T4:77.PRE EOR
%   N11:77  TT_7009_HIALM_DLY_SP  "TT-7009 HI ALARM DELAY SP FROM HMI" %
%   T4:77  TT_7009_HIALM_DLY_TM  "TT-7009 HI ALARM DELAY" %
% Rung: 82 %
SOR MOV N11:78 T4:78.PRE EOR
%   N11:78  TT_7010_LOALM_DLY_SP  "TT-7010 LO ALARM DELAY SP FROM HMI" %
%   T4:78  TT_7010_LOALM_DLY_TM  "TT-7010 LO ALARM DELAY" %
% Rung: 83 %
SOR MOV N11:79 T4:79.PRE EOR
%   N11:79  TT_7010_HIALM_DLY_SP  "TT-7010 HI ALARM DELAY SP FROM HMI" %
%   T4:79  TT_7010_HIALM_DLY_TM  "TT-7010 HI ALARM DELAY" %
% Rung: 84 %
SOR MOV N11:80 T4:80.PRE EOR
%   N11:80  TT_7020_LOALM_DLY_SP  "TT-7020 LO ALARM DELAY SP FROM HMI" %
%   T4:80  TT_7020_LOALM_DLY_TM  "TT-7020 LO ALARM DELAY" %
% Rung: 85 %
SOR MOV N11:81 T4:81.PRE EOR
%   N11:81  TT_7020_HIALM_DLY_SP  "TT-7020 HI ALARM DELAY SP FROM HMI" %
%   T4:81  TT_7020_HIALM_DLY_TM  "TT-7020 HI ALARM DELAY" %
% Rung: 86 %
SOR MOV N11:82 T4:82.PRE EOR
%   N11:82  TT_7000_LOALM_DLY_SP  "TT-7000 LO ALARM DELAY SP FROM HMI" %
%   T4:82  TT_7000_LOALM_DLY_TM  "TT-7000 LO ALARM DELAY" %
% Rung: 87 %
SOR MOV N11:83 T4:83.PRE EOR
%   N11:83  TT_7000_HIALM_DLY_SP  "TT-7000 HI ALARM DELAY SP FROM HMI" %
%   T4:83  TT_7000_HIALM_DLY_TM  "TT-7000 HI ALARM DELAY" %

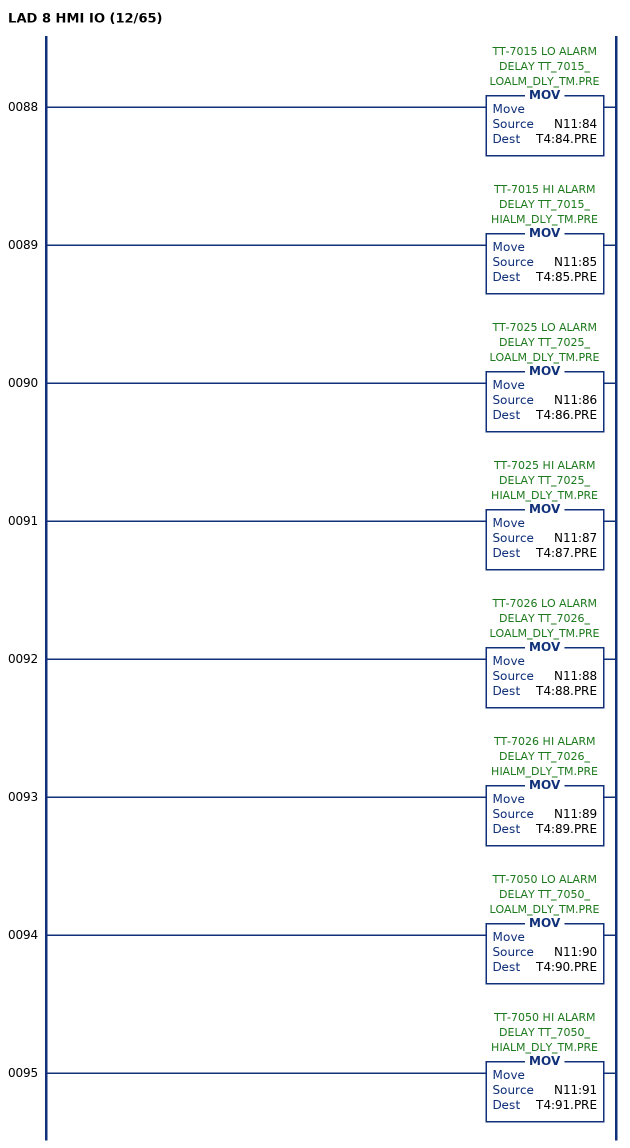
% Rung: 88 %
SOR MOV N11:84 T4:84.PRE EOR
%   N11:84  TT_7015_LOALM_DLY_SP  "TT-7015 LO ALARM DELAY SP FROM HMI" %
%   T4:84  TT_7015_LOALM_DLY_TM  "TT-7015 LO ALARM DELAY" %
% Rung: 89 %
SOR MOV N11:85 T4:85.PRE EOR
%   N11:85  TT_7015_HIALM_DLY_SP  "TT-7015 HI ALARM DELAY SP FROM HMI" %
%   T4:85  TT_7015_HIALM_DLY_TM  "TT-7015 HI ALARM DELAY" %
% Rung: 90 %
SOR MOV N11:86 T4:86.PRE EOR
%   N11:86  TT_7025_LOALM_DLY_SP  "TT-7025 LO ALARM DELAY SP FROM HMI" %
%   T4:86  TT_7025_LOALM_DLY_TM  "TT-7025 LO ALARM DELAY" %
% Rung: 91 %
SOR MOV N11:87 T4:87.PRE EOR
%   N11:87  TT_7025_HIALM_DLY_SP  "TT-7025 HI ALARM DELAY SP FROM HMI" %
%   T4:87  TT_7025_HIALM_DLY_TM  "TT-7025 HI ALARM DELAY" %
% Rung: 92 %
SOR MOV N11:88 T4:88.PRE EOR
%   N11:88  TT_7026_LOALM_DLY_SP  "TT-7026 LO ALARM DELAY SP FROM HMI" %
%   T4:88  TT_7026_LOALM_DLY_TM  "TT-7026 LO ALARM DELAY" %
% Rung: 93 %
SOR MOV N11:89 T4:89.PRE EOR
%   N11:89  TT_7026_HIALM_DLY_SP  "TT-7026 HI ALARM DELAY SP FROM HMI" %
%   T4:89  TT_7026_HIALM_DLY_TM  "TT-7026 HI ALARM DELAY" %
% Rung: 94 %
SOR MOV N11:90 T4:90.PRE EOR
%   N11:90  TT_7050_LOALM_DLY_SP  "TT-7050 LO ALARM DELAY SP FROM HMI" %
%   T4:90  TT_7050_LOALM_DLY_TM  "TT-7050 LO ALARM DELAY" %
% Rung: 95 %
SOR MOV N11:91 T4:91.PRE EOR
%   N11:91  TT_7050_HIALM_DLY_SP  "TT-7050 HI ALARM DELAY SP FROM HMI" %
%   T4:91  TT_7050_HIALM_DLY_TM  "TT-7050 HI ALARM DELAY" %

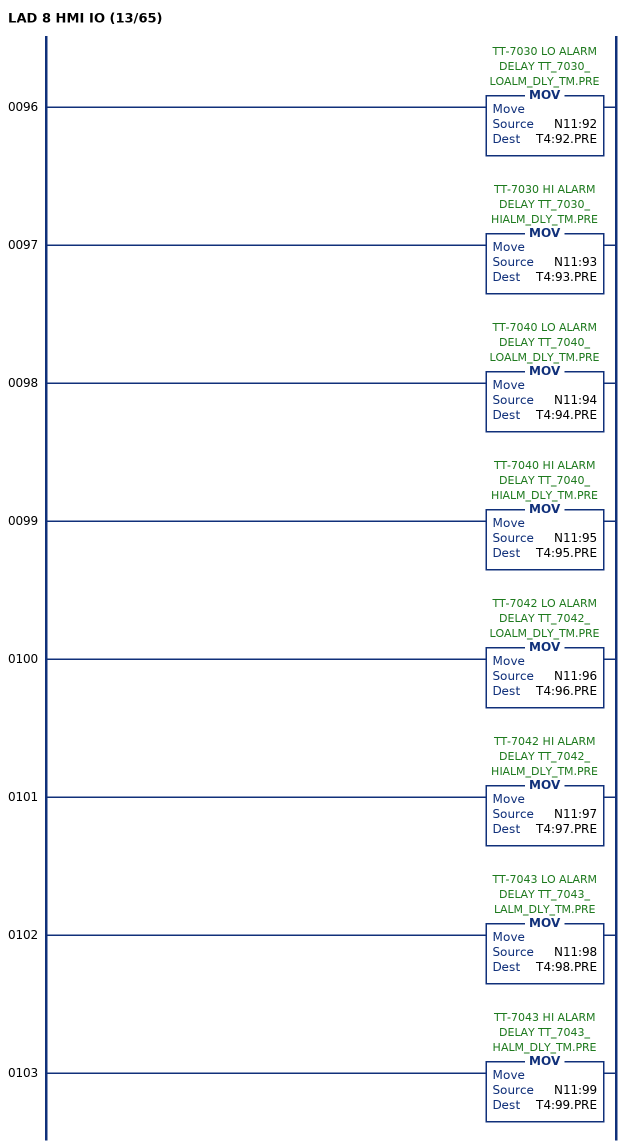
% Rung: 96 %
SOR MOV N11:92 T4:92.PRE EOR
%   N11:92  TT_7030_LOALM_DLY_SP  "TT-7030 LO ALARM DELAY SP FROM HMI" %
%   T4:92  TT_7030_LOALM_DLY_TM  "TT-7030 LO ALARM DELAY" %
% Rung: 97 %
SOR MOV N11:93 T4:93.PRE EOR
%   N11:93  TT_7030_HIALM_DLY_SP  "TT-7030 HI ALARM DELAY SP FROM HMI" %
%   T4:93  TT_7030_HIALM_DLY_TM  "TT-7030 HI ALARM DELAY" %
% Rung: 98 %
SOR MOV N11:94 T4:94.PRE EOR
%   N11:94  TT_7040_LOALM_DLY_SP  "TT-7040 LO ALARM DELAY SP FROM HMI" %
%   T4:94  TT_7040_LOALM_DLY_TM  "TT-7040 LO ALARM DELAY" %
% Rung: 99 %
SOR MOV N11:95 T4:95.PRE EOR
%   N11:95  TT_7040_HIALM_DLY_SP  "TT-7040 HI ALARM DELAY SP FROM HMI" %
%   T4:95  TT_7040_HIALM_DLY_TM  "TT-7040 HI ALARM DELAY" %
% Rung: 100 %
SOR MOV N11:96 T4:96.PRE EOR
%   N11:96  TT_7042_LOALM_DLY_SP  "TT-7042 LO ALARM DELAY SP FROM HMI" %
%   T4:96  TT_7042_LOALM_DLY_TM  "TT-7042 LO ALARM DELAY" %
% Rung: 101 %
SOR MOV N11:97 T4:97.PRE EOR
%   N11:97  TT_7042_HIALM_DLY_SP  "TT-7042 HI ALARM DELAY SP FROM HMI" %
%   T4:97  TT_7042_HIALM_DLY_TM  "TT-7042 HI ALARM DELAY" %
% Rung: 102 %
SOR MOV N11:98 T4:98.PRE EOR
%   N11:98  TT_7043_LALM_DLY_SP  "TT-7043 LO ALARM DELAY SP FROM HMI" %
%   T4:98  TT_7043_LALM_DLY_TM  "TT-7043 LO ALARM DELAY" %
% Rung: 103 %
SOR MOV N11:99 T4:99.PRE EOR
%   N11:99  TT_7043_HALM_DLY_SP  "TT-7043 HI ALARM DELAY SP FROM HMI" %
%   T4:99  TT_7043_HALM_DLY_TM  "TT-7043 HI ALARM DELAY" %

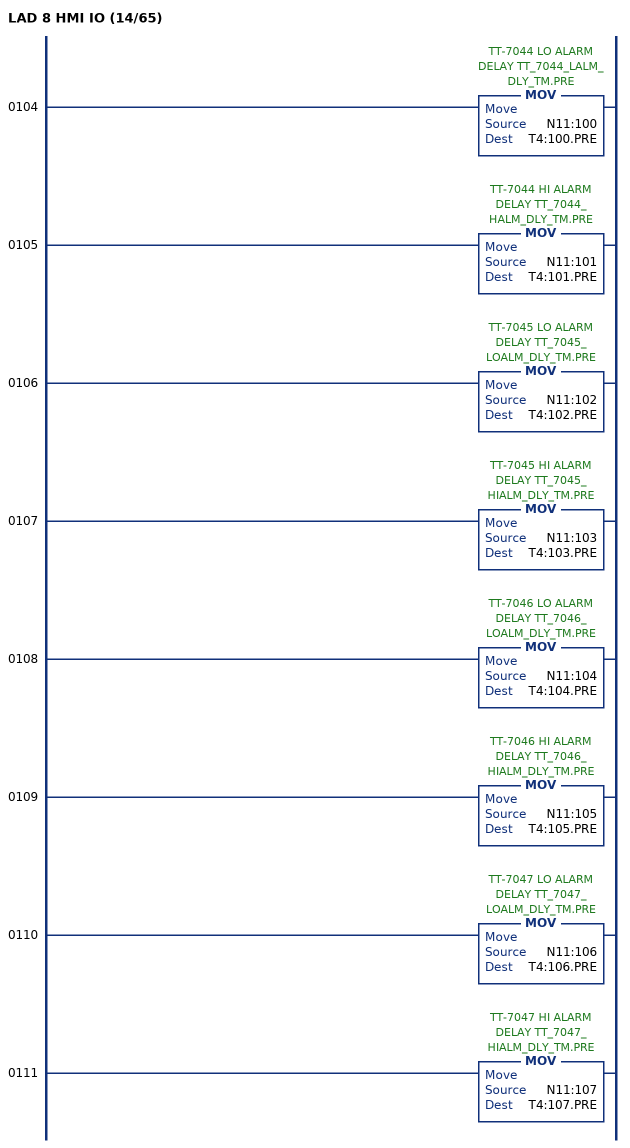
% Rung: 104 %
SOR MOV N11:100 T4:100.PRE EOR
%   N11:100  TT_7044_LALM_DLY_SP  "TT-7044 LO ALARM DELAY SP FROM HMI" %
%   T4:100  TT_7044_LALM_DLY_TM  "TT-7044 LO ALARM DELAY" %
% Rung: 105 %
SOR MOV N11:101 T4:101.PRE EOR
%   N11:101  TT_7044_HALM_DLY_SP  "TT-7044 HI ALARM DELAY SP FROM HMI" %
%   T4:101  TT_7044_HALM_DLY_TM  "TT-7044 HI ALARM DELAY" %
% Rung: 106 %
SOR MOV N11:102 T4:102.PRE EOR
%   N11:102  TT_7045_LOALM_DLY_SP  "TT-7045 LO ALARM DELAY SP FROM HMI" %
%   T4:102  TT_7045_LOALM_DLY_TM  "TT-7045 LO ALARM DELAY" %
% Rung: 107 %
SOR MOV N11:103 T4:103.PRE EOR
%   N11:103  TT_7045_HIALM_DLY_SP  "TT-7045 HI ALARM DELAY SP FROM HMI" %
%   T4:103  TT_7045_HIALM_DLY_TM  "TT-7045 HI ALARM DELAY" %
% Rung: 108 %
SOR MOV N11:104 T4:104.PRE EOR
%   N11:104  TT_7046_LOALM_DLY_SP  "TT-7046 LO ALARM DELAY SP FROM HMI" %
%   T4:104  TT_7046_LOALM_DLY_TM  "TT-7046 LO ALARM DELAY" %
% Rung: 109 %
SOR MOV N11:105 T4:105.PRE EOR
%   N11:105  TT_7046_HIALM_DLY_SP  "TT-7046 HI ALARM DELAY SP FROM HMI" %
%   T4:105  TT_7046_HIALM_DLY_TM  "TT-7046 HI ALARM DELAY" %
% Rung: 110 %
SOR MOV N11:106 T4:106.PRE EOR
%   N11:106  TT_7047_LOALM_DLY_SP  "TT-7047 LO ALARM DELAY SP FROM HMI" %
%   T4:106  TT_7047_LOALM_DLY_TM  "TT-7047 LO ALARM DELAY" %
% Rung: 111 %
SOR MOV N11:107 T4:107.PRE EOR
%   N11:107  TT_7047_HIALM_DLY_SP  "TT-7047 HI ALARM DELAY SP FROM HMI" %
%   T4:107  TT_7047_HIALM_DLY_TM  "TT-7047 HI ALARM DELAY" %

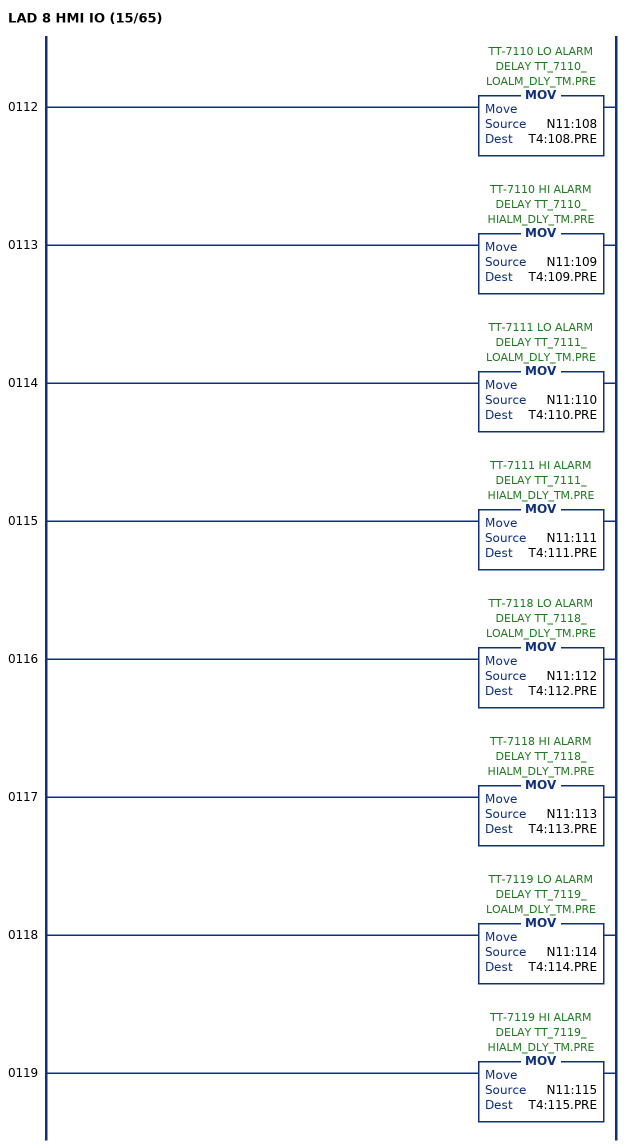
% Rung: 112 %
SOR MOV N11:108 T4:108.PRE EOR
%   N11:108  TT_7110_LOALM_DLY_SP  "TT-7110 LO ALARM DELAY SP FROM HMI" %
%   T4:108  TT_7110_LOALM_DLY_TM  "TT-7110 LO ALARM DELAY" %
% Rung: 113 %
SOR MOV N11:109 T4:109.PRE EOR
%   N11:109  TT_7110_HIALM_DLY_SP  "TT-7110 HI ALARM DELAY SP FROM HMI" %
%   T4:109  TT_7110_HIALM_DLY_TM  "TT-7110 HI ALARM DELAY" %
% Rung: 114 %
SOR MOV N11:110 T4:110.PRE EOR
%   N11:110  TT_7111_LOALM_DLY_SP  "TT-7111 LO ALARM DELAY SP FROM HMI" %
%   T4:110  TT_7111_LOALM_DLY_TM  "TT-7111 LO ALARM DELAY" %
% Rung: 115 %
SOR MOV N11:111 T4:111.PRE EOR
%   N11:111  TT_7111_HIALM_DLY_SP  "TT-7111 HI ALARM DELAY SP FROM HMI" %
%   T4:111  TT_7111_HIALM_DLY_TM  "TT-7111 HI ALARM DELAY" %
% Rung: 116 %
SOR MOV N11:112 T4:112.PRE EOR
%   N11:112  TT_7118_LOALM_DLY_SP  "TT-7118 LO ALARM DELAY SP FROM HMI" %
%   T4:112  TT_7118_LOALM_DLY_TM  "TT-7118 LO ALARM DELAY" %
% Rung: 117 %
SOR MOV N11:113 T4:113.PRE EOR
%   N11:113  TT_7118_HIALM_DLY_SP  "TT-7118 HI ALARM DELAY SP FROM HMI" %
%   T4:113  TT_7118_HIALM_DLY_TM  "TT-7118 HI ALARM DELAY" %
% Rung: 118 %
SOR MOV N11:114 T4:114.PRE EOR
%   N11:114  TT_7119_LOALM_DLY_SP  "TT-7119 LO ALARM DELAY SP FROM HMI" %
%   T4:114  TT_7119_LOALM_DLY_TM  "TT-7119 LO ALARM DELAY" %
% Rung: 119 %
SOR MOV N11:115 T4:115.PRE EOR
%   N11:115  TT_7119_HIALM_DLY_SP  "TT-7119 HI ALARM DELAY SP FROM HMI" %
%   T4:115  TT_7119_HIALM_DLY_TM  "TT-7119 HI ALARM DELAY" %

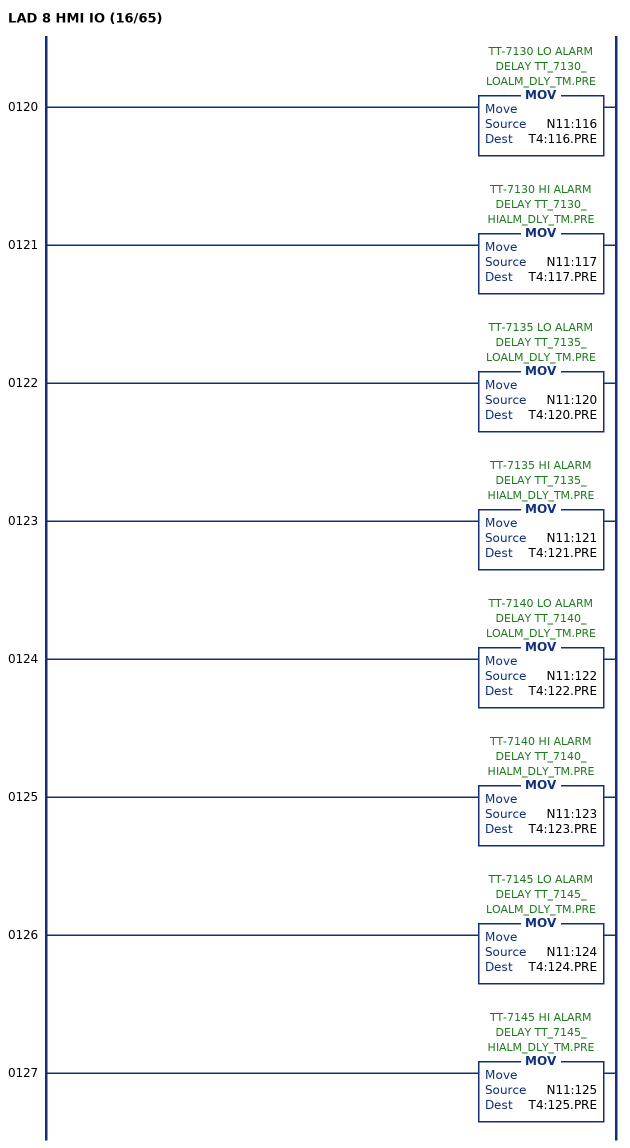
% Rung: 120 %
SOR MOV N11:116 T4:116.PRE EOR
%   N11:116  TT_7130_LOALM_DLY_SP  "TT-7130 LO ALARM DELAY SP FROM HMI" %
%   T4:116  TT_7130_LOALM_DLY_TM  "TT-7130 LO ALARM DELAY" %
% Rung: 121 %
SOR MOV N11:117 T4:117.PRE EOR
%   N11:117  TT_7130_HIALM_DLY_SP  "TT-7130 HI ALARM DELAY SP FROM HMI" %
%   T4:117  TT_7130_HIALM_DLY_TM  "TT-7130 HI ALARM DELAY" %
% Rung: 122 %
SOR MOV N11:120 T4:120.PRE EOR
%   N11:120  TT_7135_LOALM_DLY_SP  "TT-7135 LO ALARM DELAY SP FROM HMI" %
%   T4:120  TT_7135_LOALM_DLY_TM  "TT-7135 LO ALARM DELAY" %
% Rung: 123 %
SOR MOV N11:121 T4:121.PRE EOR
%   N11:121  TT_7135_HIALM_DLY_SP  "TT-7135 HI ALARM DELAY SP FROM HMI" %
%   T4:121  TT_7135_HIALM_DLY_TM  "TT-7135 HI ALARM DELAY" %
% Rung: 124 %
SOR MOV N11:122 T4:122.PRE EOR
%   N11:122  TT_7140_LOALM_DLY_SP  "TT-7140 LO ALARM DELAY SP FROM HMI" %
%   T4:122  TT_7140_LOALM_DLY_TM  "TT-7140 LO ALARM DELAY" %
% Rung: 125 %
SOR MOV N11:123 T4:123.PRE EOR
%   N11:123  TT_7140_HIALM_DLY_SP  "TT-7140 HI ALARM DELAY SP FROM HMI" %
%   T4:123  TT_7140_HIALM_DLY_TM  "TT-7140 HI ALARM DELAY" %
% Rung: 126 %
SOR MOV N11:124 T4:124.PRE EOR
%   N11:124  TT_7145_LOALM_DLY_SP  "TT-7145 LO ALARM DELAY SP FROM HMI" %
%   T4:124  TT_7145_LOALM_DLY_TM  "TT-7145 LO ALARM DELAY" %
% Rung: 127 %
SOR MOV N11:125 T4:125.PRE EOR
%   N11:125  TT_7145_HIALM_DLY_SP  "TT-7145 HI ALARM DELAY SP FROM HMI" %
%   T4:125  TT_7145_HIALM_DLY_TM  "TT-7145 HI ALARM DELAY" %

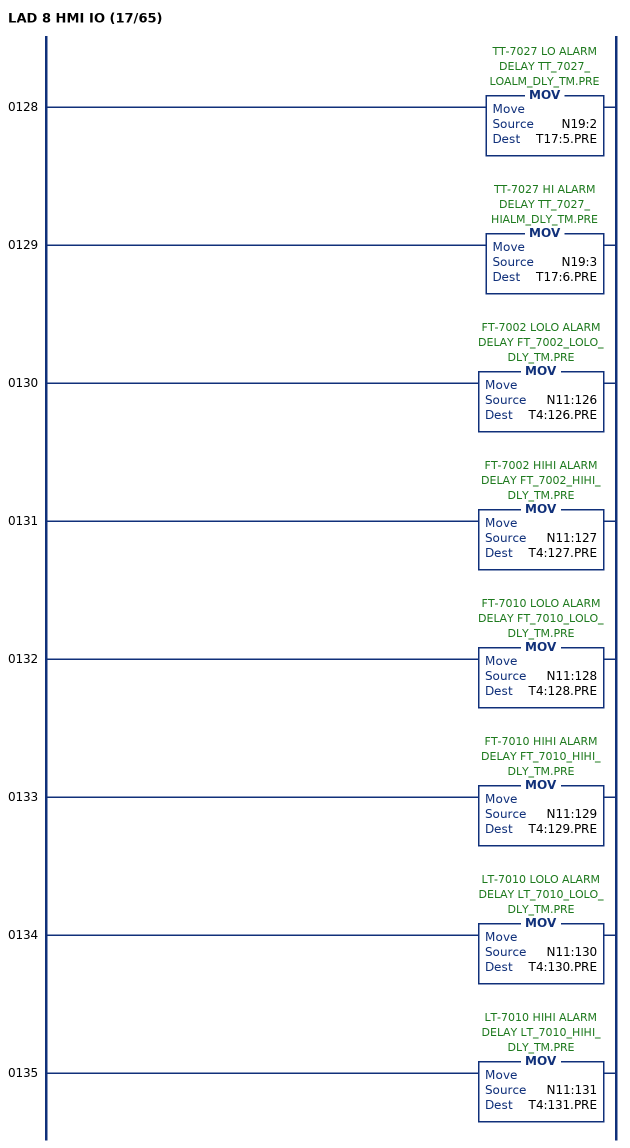
% Rung: 128 %
SOR MOV N19:2 T17:5.PRE EOR
%   N19:2  TT_7027_LOALM_DLY_SP  "TT-7027 LO ALARM DELAY SP FROM HMI" %
%   T17:5  TT_7027_LOALM_DLY_TM  "TT-7027 LO ALARM DELAY" %
% Rung: 129 %
SOR MOV N19:3 T17:6.PRE EOR
%   N19:3  TT_7027_HIALM_DLY_SP  "TT-7027 HI ALARM DELAY SP FROM HMI" %
%   T17:6  TT_7027_HIALM_DLY_TM  "TT-7027 HI ALARM DELAY" %
% Rung: 130 %
SOR MOV N11:126 T4:126.PRE EOR
%   N11:126  FT_7002_LOLO_DLY_SP  "FT-7002 LOLO ALARM DELAY SP FROM HMI" %
%   T4:126  FT_7002_LOLO_DLY_TM  "FT-7002 LOLO ALARM DELAY" %
% Rung: 131 %
SOR MOV N11:127 T4:127.PRE EOR
%   N11:127  FT_7002_HIHI_DLY_SP  "FT-7002 HIHI ALARM DELAY SP FROM HMI" %
%   T4:127  FT_7002_HIHI_DLY_TM  "FT-7002 HIHI ALARM DELAY" %
% Rung: 132 %
SOR MOV N11:128 T4:128.PRE EOR
%   N11:128  FT_7010_LOLO_DLY_SP  "FT-7010 LOLO ALARM DELAY SP FROM HMI" %
%   T4:128  FT_7010_LOLO_DLY_TM  "FT-7010 LOLO ALARM DELAY" %
% Rung: 133 %
SOR MOV N11:129 T4:129.PRE EOR
%   N11:129  FT_7010_HIHI_DLY_SP  "FT-7010 HIHI ALARM DELAY SP FROM HMI" %
%   T4:129  FT_7010_HIHI_DLY_TM  "FT-7010 HIHI ALARM DELAY" %
% Rung: 134 %
SOR MOV N11:130 T4:130.PRE EOR
%   N11:130  LT_7010_LOLO_DLY_SP  "LT-7010 LOLO ALARM DELAY SP FROM HMI" %
%   T4:130  LT_7010_LOLO_DLY_TM  "LT-7010 LOLO ALARM DELAY" %
% Rung: 135 %
SOR MOV N11:131 T4:131.PRE EOR
%   N11:131  LT_7010_HIHI_DLY_SP  "LT-7010 HIHI ALARM DELAY SP FROM HMI" %
%   T4:131  LT_7010_HIHI_DLY_TM  "LT-7010 HIHI ALARM DELAY" %

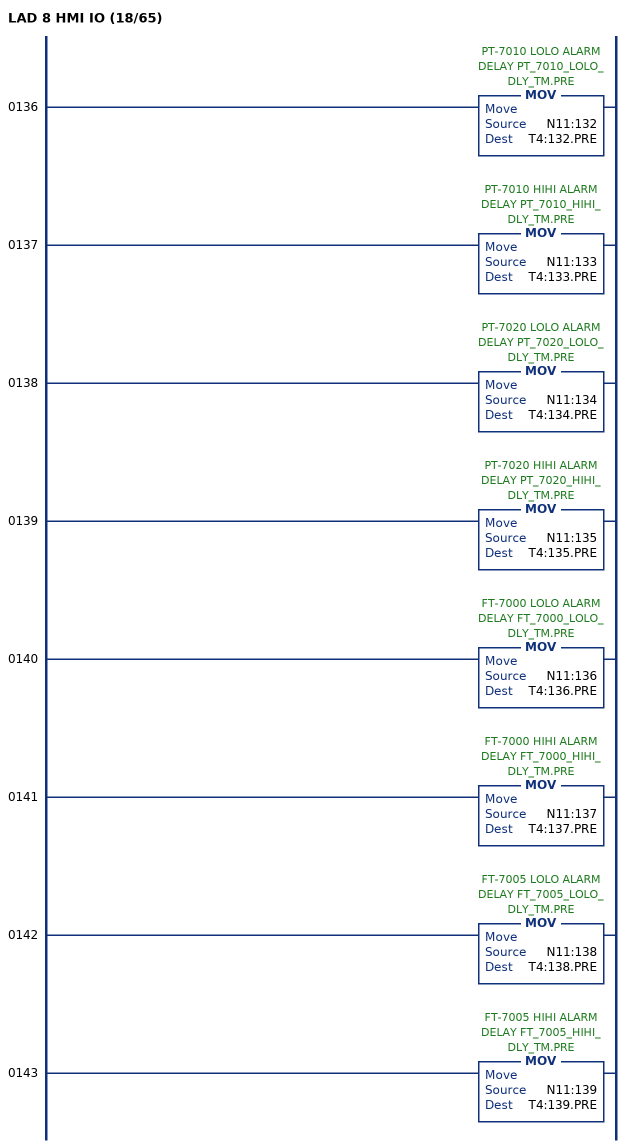
% Rung: 136 %
SOR MOV N11:132 T4:132.PRE EOR
%   N11:132  PT_7010_LOLO_DLY_SP  "PT-7010 LOLO ALARM DELAY SP FROM HMI" %
%   T4:132  PT_7010_LOLO_DLY_TM  "PT-7010 LOLO ALARM DELAY" %
% Rung: 137 %
SOR MOV N11:133 T4:133.PRE EOR
%   N11:133  PT_7010_HIHI_DLY_SP  "PT-7010 HIHI ALARM DELAY SP FROM HMI" %
%   T4:133  PT_7010_HIHI_DLY_TM  "PT-7010 HIHI ALARM DELAY" %
% Rung: 138 %
SOR MOV N11:134 T4:134.PRE EOR
%   N11:134  PT_7020_LOLO_DLY_SP  "PT-7020 LOLO ALARM DELAY SP FROM HMI" %
%   T4:134  PT_7020_LOLO_DLY_TM  "PT-7020 LOLO ALARM DELAY" %
% Rung: 139 %
SOR MOV N11:135 T4:135.PRE EOR
%   N11:135  PT_7020_HIHI_DLY_SP  "PT-7020 HIHI ALARM DELAY SP FROM HMI" %
%   T4:135  PT_7020_HIHI_DLY_TM  "PT-7020 HIHI ALARM DELAY" %
% Rung: 140 %
SOR MOV N11:136 T4:136.PRE EOR
%   N11:136  FT_7000_LOLO_DLY_SP  "FT-7000 LOLO ALARM DELAY SP FROM HMI" %
%   T4:136  FT_7000_LOLO_DLY_TM  "FT-7000 LOLO ALARM DELAY" %
% Rung: 141 %
SOR MOV N11:137 T4:137.PRE EOR
%   N11:137  FT_7000_HIHI_DLY_SP  "FT-7000 HIHI ALARM DELAY SP FROM HMI" %
%   T4:137  FT_7000_HIHI_DLY_TM  "FT-7000 HIHI ALARM DELAY" %
% Rung: 142 %
SOR MOV N11:138 T4:138.PRE EOR
%   N11:138  FT_7005_LOLO_DLY_SP  "FT-7005 LOLO ALARM DELAY SP FROM HMI" %
%   T4:138  FT_7005_LOLO_DLY_TM  "FT-7005 LOLO ALARM DELAY" %
% Rung: 143 %
SOR MOV N11:139 T4:139.PRE EOR
%   N11:139  FT_7005_HIHI_DLY_SP  "FT-7005 HIHI ALARM DELAY SP FROM HMI" %
%   T4:139  FT_7005_HIHI_DLY_TM  "FT-7005 HIHI ALARM DELAY" %

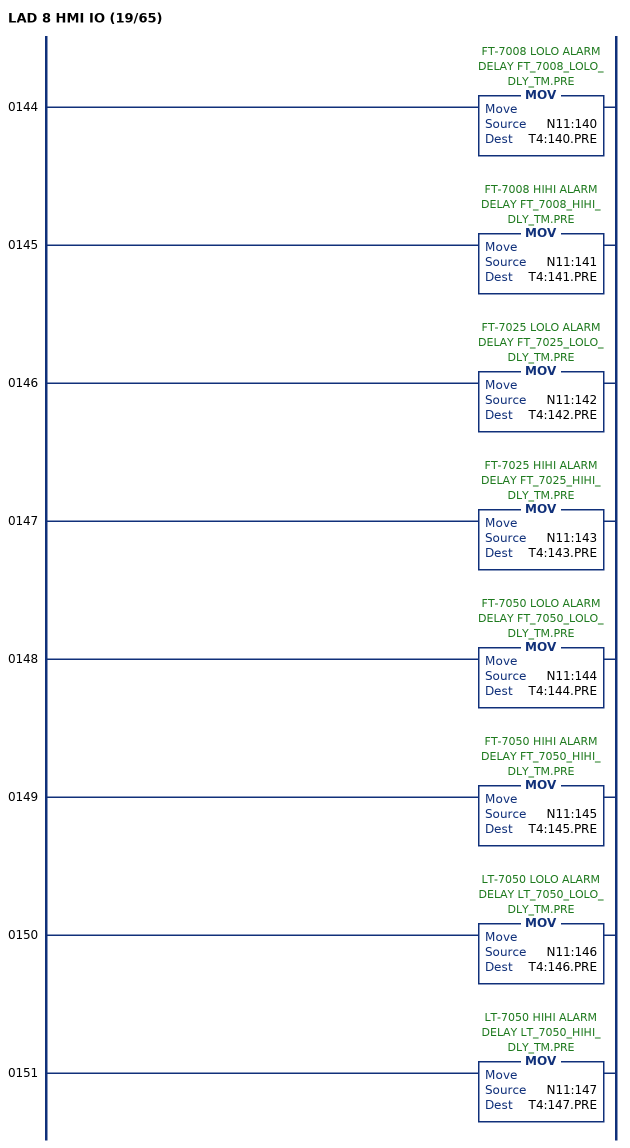
% Rung: 144 %
SOR MOV N11:140 T4:140.PRE EOR
%   N11:140  FT_7008_LOLO_DLY_SP  "FT-7008 LOLO ALARM DELAY SP FROM HMI" %
%   T4:140  FT_7008_LOLO_DLY_TM  "FT-7008 LOLO ALARM DELAY" %
% Rung: 145 %
SOR MOV N11:141 T4:141.PRE EOR
%   N11:141  FT_7008_HIHI_DLY_SP  "FT-7008 HIHI ALARM DELAY SP FROM HMI" %
%   T4:141  FT_7008_HIHI_DLY_TM  "FT-7008 HIHI ALARM DELAY" %
% Rung: 146 %
SOR MOV N11:142 T4:142.PRE EOR
%   N11:142  FT_7025_LOLO_DLY_SP  "FT-7025 LOLO ALARM DELAY SP FROM HMI" %
%   T4:142  FT_7025_LOLO_DLY_TM  "FT-7025 LOLO ALARM DELAY" %
% Rung: 147 %
SOR MOV N11:143 T4:143.PRE EOR
%   N11:143  FT_7025_HIHI_DLY_SP  "FT-7025 HIHI ALARM DELAY SP FROM HMI" %
%   T4:143  FT_7025_HIHI_DLY_TM  "FT-7025 HIHI ALARM DELAY" %
% Rung: 148 %
SOR MOV N11:144 T4:144.PRE EOR
%   N11:144  FT_7050_LOLO_DLY_SP  "FT-7050 LOLO ALARM DELAY SP FROM HMI" %
%   T4:144  FT_7050_LOLO_DLY_TM  "FT-7050 LOLO ALARM DELAY" %
% Rung: 149 %
SOR MOV N11:145 T4:145.PRE EOR
%   N11:145  FT_7050_HIHI_DLY_SP  "FT-7050 HIHI ALARM DELAY SP FROM HMI" %
%   T4:145  FT_7050_HIHI_DLY_TM  "FT-7050 HIHI ALARM DELAY" %
% Rung: 150 %
SOR MOV N11:146 T4:146.PRE EOR
%   N11:146  LT_7050_LOLO_DLY_SP  "LT-7050 LOLO ALARM DELAY SP FROM HMI" %
%   T4:146  LT_7050_LOLO_DLY_TM  "LT-7050 LOLO ALARM DELAY" %
% Rung: 151 %
SOR MOV N11:147 T4:147.PRE EOR
%   N11:147  LT_7050_HIHI_DLY_SP  "LT-7050 HIHI ALARM DELAY SP FROM HMI" %
%   T4:147  LT_7050_HIHI_DLY_TM  "LT-7050 HIHI ALARM DELAY" %

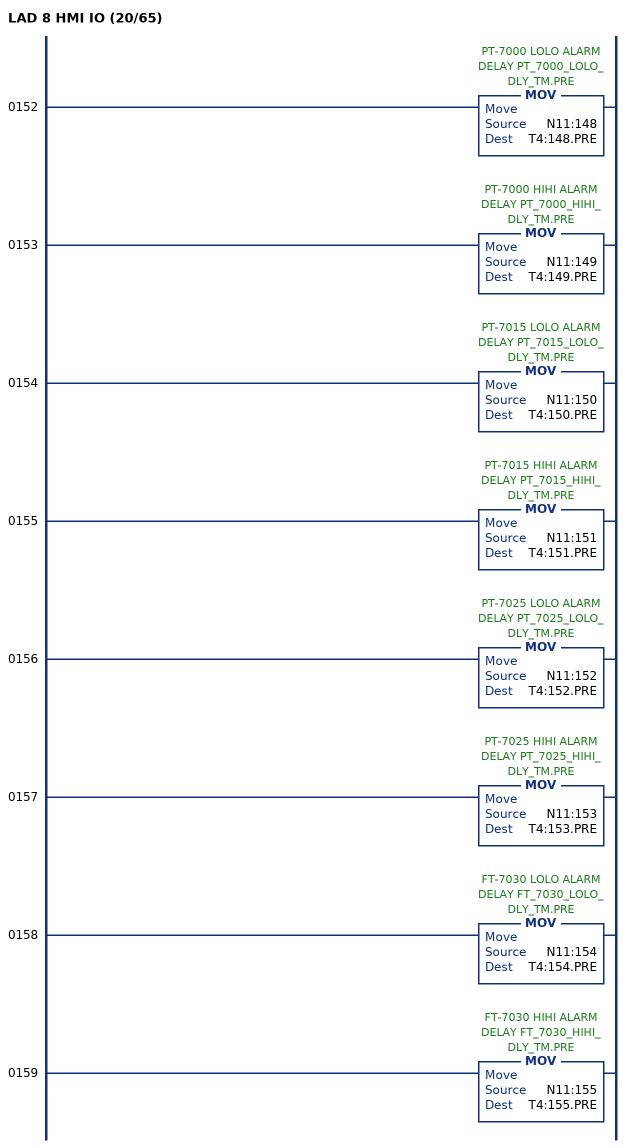
% Rung: 152 %
SOR MOV N11:148 T4:148.PRE EOR
%   N11:148  PT_7000_LOLO_DLY_SP  "PT-7000 LOLO ALARM DELAY SP FROM HMI" %
%   T4:148  PT_7000_LOLO_DLY_TM  "PT-7000 LOLO ALARM DELAY" %
% Rung: 153 %
SOR MOV N11:149 T4:149.PRE EOR
%   N11:149  PT_7000_HIHI_DLY_SP  "PT-7000 HIHI ALARM DELAY SP FROM HMI" %
%   T4:149  PT_7000_HIHI_DLY_TM  "PT-7000 HIHI ALARM DELAY" %
% Rung: 154 %
SOR MOV N11:150 T4:150.PRE EOR
%   N11:150  PT_7015_LOLO_DLY_SP  "PT-7015 LOLO ALARM DELAY SP FROM HMI" %
%   T4:150  PT_7015_LOLO_DLY_TM  "PT-7015 LOLO ALARM DELAY" %
% Rung: 155 %
SOR MOV N11:151 T4:151.PRE EOR
%   N11:151  PT_7015_HIHI_DLY_SP  "PT-7015 HIHI ALARM DELAY SP FROM HMI" %
%   T4:151  PT_7015_HIHI_DLY_TM  "PT-7015 HIHI ALARM DELAY" %
% Rung: 156 %
SOR MOV N11:152 T4:152.PRE EOR
%   N11:152  PT_7025_LOLO_DLY_SP  "PT-7025 LOLO ALARM DELAY SP FROM HMI" %
%   T4:152  PT_7025_LOLO_DLY_TM  "PT-7025 LOLO ALARM DELAY" %
% Rung: 157 %
SOR MOV N11:153 T4:153.PRE EOR
%   N11:153  PT_7025_HIHI_DLY_SP  "PT-7025 HIHI ALARM DELAY SP FROM HMI" %
%   T4:153  PT_7025_HIHI_DLY_TM  "PT-7025 HIHI ALARM DELAY" %
% Rung: 158 %
SOR MOV N11:154 T4:154.PRE EOR
%   N11:154  FT_7030_LOLO_DLY_SP  "FT-7030 LOLO ALARM DELAY SP FROM HMI" %
%   T4:154  FT_7030_LOLO_DLY_TM  "FT-7030 LOLO ALARM DELAY" %
% Rung: 159 %
SOR MOV N11:155 T4:155.PRE EOR
%   N11:155  FT_7030_HIHI_DLY_SP  "FT-7030 HIHI ALARM DELAY SP FROM HMI" %
%   T4:155  FT_7030_HIHI_DLY_TM  "FT-7030 HIHI ALARM DELAY" %

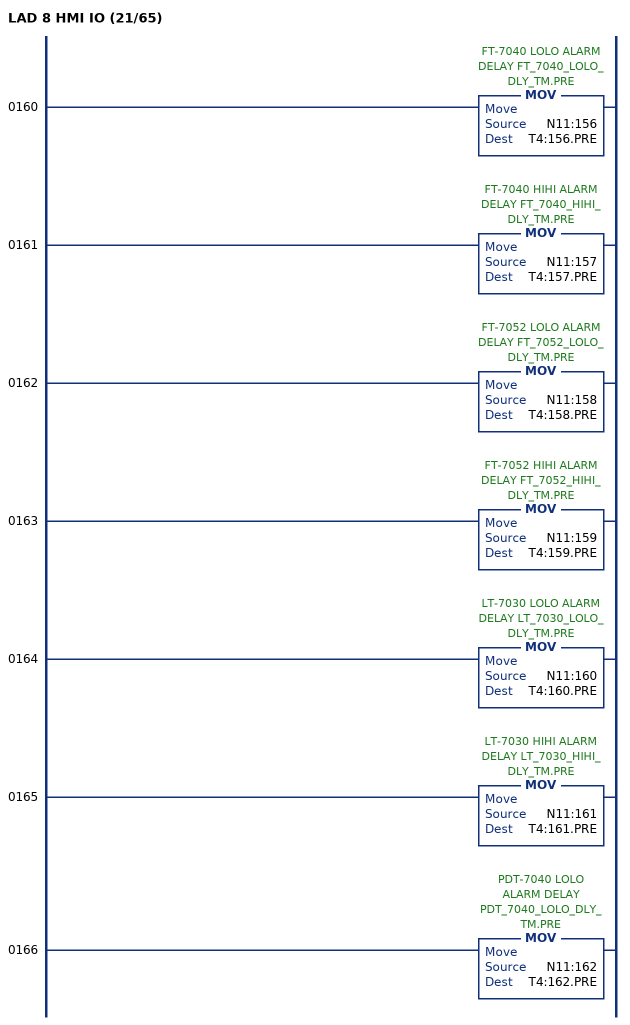
% Rung: 160 %
SOR MOV N11:156 T4:156.PRE EOR
%   N11:156  FT_7040_LOLO_DLY_SP  "FT-7040 LOLO ALARM DELAY SP FROM HMI" %
%   T4:156  FT_7040_LOLO_DLY_TM  "FT-7040 LOLO ALARM DELAY" %
% Rung: 161 %
SOR MOV N11:157 T4:157.PRE EOR
%   N11:157  FT_7040_HIHI_DLY_SP  "FT-7040 HIHI ALARM DELAY SP FROM HMI" %
%   T4:157  FT_7040_HIHI_DLY_TM  "FT-7040 HIHI ALARM DELAY" %
% Rung: 162 %
SOR MOV N11:158 T4:158.PRE EOR
%   N11:158  FT_7052_LOLO_DLY_SP  "FT-7052 LOLO ALARM DELAY SP FROM HMI" %
%   T4:158  FT_7052_LOLO_DLY_TM  "FT-7052 LOLO ALARM DELAY" %
% Rung: 163 %
SOR MOV N11:159 T4:159.PRE EOR
%   N11:159  FT_7052_HIHI_DLY_SP  "FT-7052 HIHI ALARM DELAY SP FROM HMI" %
%   T4:159  FT_7052_HIHI_DLY_TM  "FT-7052 HIHI ALARM DELAY" %
% Rung: 164 %
SOR MOV N11:160 T4:160.PRE EOR
%   N11:160  LT_7030_LOLO_DLY_SP  "LT-7030 LOLO ALARM DELAY SP FROM HMI" %
%   T4:160  LT_7030_LOLO_DLY_TM  "LT-7030 LOLO ALARM DELAY" %
% Rung: 165 %
SOR MOV N11:161 T4:161.PRE EOR
%   N11:161  LT_7030_HIHI_DLY_SP  "LT-7030 HIHI ALARM DELAY SP FROM HMI" %
%   T4:161  LT_7030_HIHI_DLY_TM  "LT-7030 HIHI ALARM DELAY" %
% Rung: 166 %
SOR MOV N11:162 T4:162.PRE EOR
%   N11:162  PDT_7040_LOLO_DLY_SP  "PDT-7040 LOLO ALARM DELAY SP FROM HMI" %
%   T4:162  PDT_7040_LOLO_DLY_TM  "PDT-7040 LOLO ALARM DELAY" %

